// eDataMappingVarNames.powermonitor_InputField_r_EnergySupplied: 				st_Variable:= IotExtractType(monitor.powermonitor.InputField.r_EnergySupplied, 0, 0); 
// eDataMappingVarNames.powermonitor_InputField_ar_THD_AVG: 				st_Variable:= IotExtractType(monitor.powermonitor.InputField.ar_THD[0], 1, 0); 
// eDataMappingVarNames.powermonitor_InputField_ar_THD_L1: 				st_Variable:= IotExtractType(monitor.powermonitor.InputField.ar_THD[1], 1, 0); 
// eDataMappingVarNames.powermonitor_InputField_ar_THD_L2: 				st_Variable:= IotExtractType(monitor.powermonitor.InputField.ar_THD[2], 1, 0); 
// eDataMappingVarNames.powermonitor_InputField_ar_THD_L3: 				st_Variable:= IotExtractType(monitor.powermonitor.InputField.ar_THD[3], 1, 0); 
// eDataMappingVarNames.powermonitor_InputField_ar_PowerFactor_AVG: 				st_Variable:= IotExtractType(monitor.powermonitor.InputField.ar_PowerFactor[0], 2, 0); 
// eDataMappingVarNames.powermonitor_InputField_ar_PowerFactor_L1: 				st_Variable:= IotExtractType(monitor.powermonitor.InputField.ar_PowerFactor[1], 2, 0); 
// eDataMappingVarNames.powermonitor_InputField_ar_PowerFactor_L2: 				st_Variable:= IotExtractType(monitor.powermonitor.InputField.ar_PowerFactor[2], 2, 0); 
// eDataMappingVarNames.powermonitor_InputField_ar_PowerFactor_L3: 				st_Variable:= IotExtractType(monitor.powermonitor.InputField.ar_PowerFactor[3], 2, 0); 
// eDataMappingVarNames.powermonitor_InputField_ar_Current_AVG: 				st_Variable:= IotExtractType(monitor.powermonitor.InputField.ar_Current[0], 0, 1); 
// eDataMappingVarNames.powermonitor_InputField_ar_Current_L1: 				st_Variable:= IotExtractType(monitor.powermonitor.InputField.ar_Current[1], 0, 1); 
// eDataMappingVarNames.powermonitor_InputField_ar_Current_L2: 				st_Variable:= IotExtractType(monitor.powermonitor.InputField.ar_Current[2], 0, 1); 
// eDataMappingVarNames.powermonitor_InputField_ar_Current_L3: 				st_Variable:= IotExtractType(monitor.powermonitor.InputField.ar_Current[3], 0, 1); 
// eDataMappingVarNames.powermonitor_InputField_ar_Current_N: 					st_Variable:= IotExtractType(monitor.powermonitor.InputField.ar_Current[4], 0, 1); 
// eDataMappingVarNames.powermonitor_InputField_r_CurrentUnbalance: 				st_Variable:= IotExtractType(monitor.powermonitor.InputField.r_CurrentUnbalance, 1, 0); 
// eDataMappingVarNames.powermonitor_InputField_e_ACrotationStatus: 				st_Variable:= IotExtractType(monitor.powermonitor.InputField.e_ACrotationStatus, 0, 0); 
// eDataMappingVarNames.powermonitor_InputField_ar_PhaseVoltage_AVG: 				st_Variable:= IotExtractType(monitor.powermonitor.InputField.ar_PhaseVoltage[0], 1, 1); 
// eDataMappingVarNames.powermonitor_InputField_ar_PhaseVoltage_L1: 				st_Variable:= IotExtractType(monitor.powermonitor.InputField.ar_PhaseVoltage[1], 1, 1); 
// eDataMappingVarNames.powermonitor_InputField_ar_PhaseVoltage_L2: 				st_Variable:= IotExtractType(monitor.powermonitor.InputField.ar_PhaseVoltage[2], 1, 1); 
// eDataMappingVarNames.powermonitor_InputField_ar_PhaseVoltage_L3: 				st_Variable:= IotExtractType(monitor.powermonitor.InputField.ar_PhaseVoltage[3], 1, 1); 
// eDataMappingVarNames.powermonitor_InputField_ar_LineVoltage_AVG: 				st_Variable:= IotExtractType(monitor.powermonitor.InputField.ar_LineVoltage[0], 1, 1); 
// eDataMappingVarNames.powermonitor_InputField_ar_LineVoltage_L1: 				st_Variable:= IotExtractType(monitor.powermonitor.InputField.ar_LineVoltage[1], 1, 1); 
// eDataMappingVarNames.powermonitor_InputField_ar_LineVoltage_L2: 				st_Variable:= IotExtractType(monitor.powermonitor.InputField.ar_LineVoltage[2], 1, 1); 
// eDataMappingVarNames.powermonitor_InputField_ar_LineVoltage_L3: 				st_Variable:= IotExtractType(monitor.powermonitor.InputField.ar_LineVoltage[3], 1, 1); 
// eDataMappingVarNames.powermonitor_InputField_li_TimeVoltZeroCrossup: 				st_Variable:= IotExtractType(monitor.powermonitor.InputField.li_TimeVoltZeroCrossup, 0, 0); 
// eDataMappingVarNames.powermonitor_InputField_ar_Frequency_AVG: 				st_Variable:= IotExtractType(monitor.powermonitor.InputField.ar_Frequency[0], 2, 1); 
// eDataMappingVarNames.powermonitor_InputField_ar_Frequency_L1: 				st_Variable:= IotExtractType(monitor.powermonitor.InputField.ar_Frequency[1], 2, 1); 
// eDataMappingVarNames.powermonitor_InputField_ar_Frequency_L2: 				st_Variable:= IotExtractType(monitor.powermonitor.InputField.ar_Frequency[2], 2, 1); 
// eDataMappingVarNames.powermonitor_InputField_ar_Frequency_L3: 				st_Variable:= IotExtractType(monitor.powermonitor.InputField.ar_Frequency[3], 2, 1); 
// eDataMappingVarNames.powermonitor_InputField_r_VoltageUnbalance: 				st_Variable:= IotExtractType(monitor.powermonitor.InputField.r_VoltageUnbalance, 1, 0); 
// eDataMappingVarNames.powermonitor_InputField_r_loadshare: 				st_Variable:= IotExtractType(monitor.powermonitor.InputField.r_loadshare, 1, 0); 
// eDataMappingVarNames.powermonitor_InputField_Powerlock_1_ar_ApparentPower_AVG: 				st_Variable:= IotExtractType(monitor.powermonitor.InputField.Powerlock[1].ar_ApparentPower[0], 0, 0); 
// eDataMappingVarNames.powermonitor_InputField_Powerlock_2_ar_ApparentPower_AVG: 				st_Variable:= IotExtractType(monitor.powermonitor.InputField.Powerlock[2].ar_ApparentPower[0], 0, 0); 
// eDataMappingVarNames.powermonitor_InputField_Powerlock_1_ar_ApparentPower_L1: 				st_Variable:= IotExtractType(monitor.powermonitor.InputField.Powerlock[1].ar_ApparentPower[1], 0, 0); 
// eDataMappingVarNames.powermonitor_InputField_Powerlock_2_ar_ApparentPower_L1: 				st_Variable:= IotExtractType(monitor.powermonitor.InputField.Powerlock[2].ar_ApparentPower[1], 0, 0); 
// eDataMappingVarNames.powermonitor_InputField_Powerlock_1_ar_ApparentPower_L2: 				st_Variable:= IotExtractType(monitor.powermonitor.InputField.Powerlock[1].ar_ApparentPower[2], 0, 0); 
// eDataMappingVarNames.powermonitor_InputField_Powerlock_2_ar_ApparentPower_L2: 				st_Variable:= IotExtractType(monitor.powermonitor.InputField.Powerlock[2].ar_ApparentPower[2], 0, 0); 
// eDataMappingVarNames.powermonitor_InputField_Powerlock_1_ar_ApparentPower_L3: 				st_Variable:= IotExtractType(monitor.powermonitor.InputField.Powerlock[1].ar_ApparentPower[3], 0, 0); 
// eDataMappingVarNames.powermonitor_InputField_Powerlock_2_ar_ApparentPower_L3: 				st_Variable:= IotExtractType(monitor.powermonitor.InputField.Powerlock[2].ar_ApparentPower[3], 0, 0); 
// eDataMappingVarNames.powermonitor_InputField_Powerlock_1_ar_ReactivePower_AVG: 				st_Variable:= IotExtractType(monitor.powermonitor.InputField.Powerlock[1].ar_ReactivePower[0], 0, 0); 
// eDataMappingVarNames.powermonitor_InputField_Powerlock_2_ar_ReactivePower_AVG: 				st_Variable:= IotExtractType(monitor.powermonitor.InputField.Powerlock[2].ar_ReactivePower[0], 0, 0); 
// eDataMappingVarNames.powermonitor_InputField_Powerlock_1_ar_ReactivePower_L1: 				st_Variable:= IotExtractType(monitor.powermonitor.InputField.Powerlock[1].ar_ReactivePower[1], 0, 0); 
// eDataMappingVarNames.powermonitor_InputField_Powerlock_2_ar_ReactivePower_L1: 				st_Variable:= IotExtractType(monitor.powermonitor.InputField.Powerlock[2].ar_ReactivePower[1], 0, 0); 
// eDataMappingVarNames.powermonitor_InputField_Powerlock_1_ar_ReactivePower_L2: 				st_Variable:= IotExtractType(monitor.powermonitor.InputField.Powerlock[1].ar_ReactivePower[2], 0, 0); 
// eDataMappingVarNames.powermonitor_InputField_Powerlock_2_ar_ReactivePower_L2: 				st_Variable:= IotExtractType(monitor.powermonitor.InputField.Powerlock[2].ar_ReactivePower[2], 0, 0); 
// eDataMappingVarNames.powermonitor_InputField_Powerlock_1_ar_ReactivePower_L3: 				st_Variable:= IotExtractType(monitor.powermonitor.InputField.Powerlock[1].ar_ReactivePower[3], 0, 0); 
// eDataMappingVarNames.powermonitor_InputField_Powerlock_2_ar_ReactivePower_L3: 				st_Variable:= IotExtractType(monitor.powermonitor.InputField.Powerlock[2].ar_ReactivePower[3], 0, 0); 
// eDataMappingVarNames.powermonitor_InputField_Powerlock_1_ar_ActivePower_AVG: 				st_Variable:= IotExtractType(monitor.powermonitor.InputField.Powerlock[1].ar_ActivePower[0]	, 0, 0); 
// eDataMappingVarNames.powermonitor_InputField_Powerlock_2_ar_ActivePower_AVG: 				st_Variable:= IotExtractType(monitor.powermonitor.InputField.Powerlock[2].ar_ActivePower[0]	, 0, 0); 
// eDataMappingVarNames.powermonitor_InputField_Powerlock_1_ar_ActivePower_L1: 				st_Variable:= IotExtractType(monitor.powermonitor.InputField.Powerlock[1].ar_ActivePower[1]	, 0, 0); 
// eDataMappingVarNames.powermonitor_InputField_Powerlock_2_ar_ActivePower_L1: 				st_Variable:= IotExtractType(monitor.powermonitor.InputField.Powerlock[2].ar_ActivePower[1]	, 0, 0); 
// eDataMappingVarNames.powermonitor_InputField_Powerlock_1_ar_ActivePower_L2: 				st_Variable:= IotExtractType(monitor.powermonitor.InputField.Powerlock[1].ar_ActivePower[2]	, 0, 0); 
// eDataMappingVarNames.powermonitor_InputField_Powerlock_2_ar_ActivePower_L2: 				st_Variable:= IotExtractType(monitor.powermonitor.InputField.Powerlock[2].ar_ActivePower[2]	, 0, 0); 
// eDataMappingVarNames.powermonitor_InputField_Powerlock_1_ar_ActivePower_L3: 				st_Variable:= IotExtractType(monitor.powermonitor.InputField.Powerlock[1].ar_ActivePower[3]	, 0, 0); 
// eDataMappingVarNames.powermonitor_InputField_Powerlock_2_ar_ActivePower_L3: 				st_Variable:= IotExtractType(monitor.powermonitor.InputField.Powerlock[2].ar_ActivePower[3]	, 0, 0); 
// eDataMappingVarNames.powermonitor_InputField_Powerlock_1_r_EnergyConsumed: 				st_Variable:= IotExtractType(monitor.powermonitor.InputField.Powerlock[1].r_EnergyConsumed, 0, 	0); 
// eDataMappingVarNames.powermonitor_InputField_Powerlock_2_r_EnergyConsumed: 				st_Variable:= IotExtractType(monitor.powermonitor.InputField.Powerlock[2].r_EnergyConsumed, 0, 	0); 
// eDataMappingVarNames.powermonitor_InputField_Powerlock_1_r_EnergySupplied: 				st_Variable:= IotExtractType(monitor.powermonitor.InputField.Powerlock[1].r_EnergySupplied, 0, 	0); 
// eDataMappingVarNames.powermonitor_InputField_Powerlock_2_r_EnergySupplied: 				st_Variable:= IotExtractType(monitor.powermonitor.InputField.Powerlock[2].r_EnergySupplied, 0, 	0); 
// eDataMappingVarNames.powermonitor_InputField_Powerlock_1_ar_THD_AVG: 				st_Variable:= IotExtractType(monitor.powermonitor.InputField.Powerlock[1].ar_THD[0], 0, 0);        	
// eDataMappingVarNames.powermonitor_InputField_Powerlock_2_ar_THD_AVG: 				st_Variable:= IotExtractType(monitor.powermonitor.InputField.Powerlock[2].ar_THD[0], 0, 0);        	
// eDataMappingVarNames.powermonitor_InputField_Powerlock_1_ar_THD_L1: 				st_Variable:= IotExtractType(monitor.powermonitor.InputField.Powerlock[1].ar_THD[1], 0, 0);        	
// eDataMappingVarNames.powermonitor_InputField_Powerlock_2_ar_THD_L1: 				st_Variable:= IotExtractType(monitor.powermonitor.InputField.Powerlock[2].ar_THD[1], 0, 0);        	
// eDataMappingVarNames.powermonitor_InputField_Powerlock_1_ar_THD_L2: 				st_Variable:= IotExtractType(monitor.powermonitor.InputField.Powerlock[1].ar_THD[2], 0, 0);        	
// eDataMappingVarNames.powermonitor_InputField_Powerlock_2_ar_THD_L2: 				st_Variable:= IotExtractType(monitor.powermonitor.InputField.Powerlock[2].ar_THD[2], 0, 0);        	
// eDataMappingVarNames.powermonitor_InputField_Powerlock_1_ar_THD_L3: 				st_Variable:= IotExtractType(monitor.powermonitor.InputField.Powerlock[1].ar_THD[3], 0, 0);        	
// eDataMappingVarNames.powermonitor_InputField_Powerlock_2_ar_THD_L3: 				st_Variable:= IotExtractType(monitor.powermonitor.InputField.Powerlock[2].ar_THD[3], 0, 0);        	
// eDataMappingVarNames.powermonitor_InputField_Powerlock_1_ar_PowerFactor_AVG: 				st_Variable:= IotExtractType(monitor.powermonitor.InputField.Powerlock[1].ar_PowerFactor[0]	, 2, 0); 
// eDataMappingVarNames.powermonitor_InputField_Powerlock_2_ar_PowerFactor_AVG: 				st_Variable:= IotExtractType(monitor.powermonitor.InputField.Powerlock[2].ar_PowerFactor[0]	, 2, 0); 
// eDataMappingVarNames.powermonitor_InputField_Powerlock_1_ar_PowerFactor_L1: 				st_Variable:= IotExtractType(monitor.powermonitor.InputField.Powerlock[1].ar_PowerFactor[1]	, 2, 0); 
// eDataMappingVarNames.powermonitor_InputField_Powerlock_2_ar_PowerFactor_L1: 				st_Variable:= IotExtractType(monitor.powermonitor.InputField.Powerlock[2].ar_PowerFactor[1]	, 2, 0); 
// eDataMappingVarNames.powermonitor_InputField_Powerlock_1_ar_PowerFactor_L2: 				st_Variable:= IotExtractType(monitor.powermonitor.InputField.Powerlock[1].ar_PowerFactor[2]	, 2, 0); 
// eDataMappingVarNames.powermonitor_InputField_Powerlock_2_ar_PowerFactor_L2: 				st_Variable:= IotExtractType(monitor.powermonitor.InputField.Powerlock[2].ar_PowerFactor[2]	, 2, 0); 
// eDataMappingVarNames.powermonitor_InputField_Powerlock_1_ar_PowerFactor_L3: 				st_Variable:= IotExtractType(monitor.powermonitor.InputField.Powerlock[1].ar_PowerFactor[3]	, 2, 0); 
// eDataMappingVarNames.powermonitor_InputField_Powerlock_2_ar_PowerFactor_L3: 				st_Variable:= IotExtractType(monitor.powermonitor.InputField.Powerlock[2].ar_PowerFactor[3]	, 2, 0); 
// eDataMappingVarNames.powermonitor_InputField_Powerlock_1_ar_Current_AVG: 				st_Variable:= IotExtractType(monitor.powermonitor.InputField.Powerlock[1].ar_Current[0]			, 1, 1); 
// eDataMappingVarNames.powermonitor_InputField_Powerlock_2_ar_Current_AVG: 				st_Variable:= IotExtractType(monitor.powermonitor.InputField.Powerlock[2].ar_Current[0]			, 1, 1); 
// eDataMappingVarNames.powermonitor_InputField_Powerlock_1_ar_Current_L1: 				st_Variable:= IotExtractType(monitor.powermonitor.InputField.Powerlock[1].ar_Current[1]			, 1, 1); 
// eDataMappingVarNames.powermonitor_InputField_Powerlock_2_ar_Current_L1: 				st_Variable:= IotExtractType(monitor.powermonitor.InputField.Powerlock[2].ar_Current[1]			, 1, 1); 
// eDataMappingVarNames.powermonitor_InputField_Powerlock_1_ar_Current_L2: 				st_Variable:= IotExtractType(monitor.powermonitor.InputField.Powerlock[1].ar_Current[2]			, 1, 1); 
// eDataMappingVarNames.powermonitor_InputField_Powerlock_2_ar_Current_L2: 				st_Variable:= IotExtractType(monitor.powermonitor.InputField.Powerlock[2].ar_Current[2]			, 1, 1); 
// eDataMappingVarNames.powermonitor_InputField_Powerlock_1_ar_Current_L3: 				st_Variable:= IotExtractType(monitor.powermonitor.InputField.Powerlock[1].ar_Current[3]			, 1, 1); 
// eDataMappingVarNames.powermonitor_InputField_Powerlock_2_ar_Current_L3: 				st_Variable:= IotExtractType(monitor.powermonitor.InputField.Powerlock[2].ar_Current[3]			, 1, 1); 
// eDataMappingVarNames.powermonitor_InputField_Powerlock_1_ar_Current_N: 				st_Variable:= IotExtractType(monitor.powermonitor.InputField.Powerlock[1].ar_Current[4], 1, 1); 
// eDataMappingVarNames.powermonitor_InputField_Powerlock_2_ar_Current_N: 				st_Variable:= IotExtractType(monitor.powermonitor.InputField.Powerlock[2].ar_Current[4], 1, 1); 
// eDataMappingVarNames.powermonitor_InputField_Powerlock_1_r_CurrentUnbalance: 				st_Variable:= IotExtractType(monitor.powermonitor.InputField.Powerlock[1].r_CurrentUnbalance, 0, 0); 
// eDataMappingVarNames.powermonitor_InputField_Powerlock_2_r_CurrentUnbalance: 				st_Variable:= IotExtractType(monitor.powermonitor.InputField.Powerlock[2].r_CurrentUnbalance, 0, 0); 
// eDataMappingVarNames.powermonitor_OutputField_ar_ApparentPower_AVG: 				st_Variable:= IotExtractType(monitor.powermonitor.OutputField.ar_ApparentPower[0]	, 1, 1); 
// eDataMappingVarNames.powermonitor_OutputField_ar_ApparentPower_L1: 				st_Variable:= IotExtractType(monitor.powermonitor.OutputField.ar_ApparentPower[1]		, 1, 1); 
// eDataMappingVarNames.powermonitor_OutputField_ar_ApparentPower_L2: 				st_Variable:= IotExtractType(monitor.powermonitor.OutputField.ar_ApparentPower[2]		, 1, 1); 
// eDataMappingVarNames.powermonitor_OutputField_ar_ApparentPower_L3: 				st_Variable:= IotExtractType(monitor.powermonitor.OutputField.ar_ApparentPower[3]		, 1, 1); 
// eDataMappingVarNames.powermonitor_OutputField_ar_ReactivePower_AVG: 				st_Variable:= IotExtractType(monitor.powermonitor.OutputField.ar_ReactivePower[0]	, 1, 1); 
// eDataMappingVarNames.powermonitor_OutputField_ar_ReactivePower_L1: 				st_Variable:= IotExtractType(monitor.powermonitor.OutputField.ar_ReactivePower[1]		, 1, 1); 
// eDataMappingVarNames.powermonitor_OutputField_ar_ReactivePower_L2: 				st_Variable:= IotExtractType(monitor.powermonitor.OutputField.ar_ReactivePower[2]		, 1, 1); 
// eDataMappingVarNames.powermonitor_OutputField_ar_ReactivePower_L3: 				st_Variable:= IotExtractType(monitor.powermonitor.OutputField.ar_ReactivePower[3]		, 1, 1); 
// eDataMappingVarNames.powermonitor_OutputField_ar_ActivePower_AVG: 				st_Variable:= IotExtractType(monitor.powermonitor.OutputField.ar_ActivePower[0]			, 1, 1); 
// eDataMappingVarNames.powermonitor_OutputField_ar_ActivePower_L1: 				st_Variable:= IotExtractType(monitor.powermonitor.OutputField.ar_ActivePower[1]			, 1, 1); 
// eDataMappingVarNames.powermonitor_OutputField_ar_ActivePower_L2: 				st_Variable:= IotExtractType(monitor.powermonitor.OutputField.ar_ActivePower[2]			, 1, 1); 
// eDataMappingVarNames.powermonitor_OutputField_ar_ActivePower_L3: 				st_Variable:= IotExtractType(monitor.powermonitor.OutputField.ar_ActivePower[3]			, 1, 1); 
// eDataMappingVarNames.powermonitor_OutputField_r_EnergyConsumed: 				st_Variable:= IotExtractType(monitor.powermonitor.OutputField.r_EnergyConsumed, 0, 0); 
// eDataMappingVarNames.powermonitor_OutputField_r_EnergySupplied: 				st_Variable:= IotExtractType(monitor.powermonitor.OutputField.r_EnergySupplied, 0, 0); 
// eDataMappingVarNames.powermonitor_OutputField_ar_THD_AVG: 				st_Variable:= IotExtractType(monitor.powermonitor.OutputField.ar_THD[0], 1, 0); 
// eDataMappingVarNames.powermonitor_OutputField_ar_THD_L1: 				st_Variable:= IotExtractType(monitor.powermonitor.OutputField.ar_THD[1], 1, 0); 
// eDataMappingVarNames.powermonitor_OutputField_ar_THD_L2: 				st_Variable:= IotExtractType(monitor.powermonitor.OutputField.ar_THD[2], 1, 0); 
// eDataMappingVarNames.powermonitor_OutputField_ar_THD_L3: 				st_Variable:= IotExtractType(monitor.powermonitor.OutputField.ar_THD[3], 1, 0); 
// eDataMappingVarNames.powermonitor_OutputField_ar_PowerFactor_AVG: 				st_Variable:= IotExtractType(monitor.powermonitor.OutputField.ar_PowerFactor[0], 2, 0); 
// eDataMappingVarNames.powermonitor_OutputField_ar_PowerFactor_L1: 				st_Variable:= IotExtractType(monitor.powermonitor.OutputField.ar_PowerFactor[1], 2, 0); 
// eDataMappingVarNames.powermonitor_OutputField_ar_PowerFactor_L2: 				st_Variable:= IotExtractType(monitor.powermonitor.OutputField.ar_PowerFactor[2], 2, 0); 
// eDataMappingVarNames.powermonitor_OutputField_ar_PowerFactor_L3: 				st_Variable:= IotExtractType(monitor.powermonitor.OutputField.ar_PowerFactor[3], 2, 0); 
// eDataMappingVarNames.powermonitor_OutputField_ar_Current_AVG: 				st_Variable:= IotExtractType(monitor.powermonitor.OutputField.ar_Current[0], 1, 1); 
// eDataMappingVarNames.powermonitor_OutputField_ar_Current_L1: 				st_Variable:= IotExtractType(monitor.powermonitor.OutputField.ar_Current[1], 1, 1); 
// eDataMappingVarNames.powermonitor_OutputField_ar_Current_L2: 				st_Variable:= IotExtractType(monitor.powermonitor.OutputField.ar_Current[2], 1, 1); 
// eDataMappingVarNames.powermonitor_OutputField_ar_Current_L3: 				st_Variable:= IotExtractType(monitor.powermonitor.OutputField.ar_Current[3], 1, 1); 
// eDataMappingVarNames.powermonitor_OutputField_ar_Current_N: 				st_Variable:= IotExtractType(monitor.powermonitor.OutputField.ar_Current[4], 1, 1); 
// eDataMappingVarNames.powermonitor_OutputField_r_CurrentUnbalance: 				st_Variable:= IotExtractType(monitor.powermonitor.OutputField.r_CurrentUnbalance, 1, 0); 
// eDataMappingVarNames.powermonitor_OutputField_e_ACrotationStatus: 				st_Variable:= IotExtractType(monitor.powermonitor.OutputField.e_ACrotationStatus, 0, 0); 
// eDataMappingVarNames.powermonitor_OutputField_ar_PhaseVoltage_AVG: 				st_Variable:= IotExtractType(monitor.powermonitor.OutputField.ar_PhaseVoltage[0], 1, 1); 
// eDataMappingVarNames.powermonitor_OutputField_ar_PhaseVoltage_L1: 				st_Variable:= IotExtractType(monitor.powermonitor.OutputField.ar_PhaseVoltage[1], 1, 1); 
// eDataMappingVarNames.powermonitor_OutputField_ar_PhaseVoltage_L2: 				st_Variable:= IotExtractType(monitor.powermonitor.OutputField.ar_PhaseVoltage[2], 1, 1); 
// eDataMappingVarNames.powermonitor_OutputField_ar_PhaseVoltage_L3: 				st_Variable:= IotExtractType(monitor.powermonitor.OutputField.ar_PhaseVoltage[3], 1, 1); 
// eDataMappingVarNames.powermonitor_OutputField_ar_LineVoltage_AVG: 				st_Variable:= IotExtractType(monitor.powermonitor.OutputField.ar_LineVoltage[0]	, 1, 1); 
// eDataMappingVarNames.powermonitor_OutputField_ar_LineVoltage_L1: 				st_Variable:= IotExtractType(monitor.powermonitor.OutputField.ar_LineVoltage[1]	, 1, 1); 
// eDataMappingVarNames.powermonitor_OutputField_ar_LineVoltage_L2: 				st_Variable:= IotExtractType(monitor.powermonitor.OutputField.ar_LineVoltage[2]	, 1, 1); 
// eDataMappingVarNames.powermonitor_OutputField_ar_LineVoltage_L3: 				st_Variable:= IotExtractType(monitor.powermonitor.OutputField.ar_LineVoltage[3]	, 1, 1); 
// eDataMappingVarNames.powermonitor_OutputField_li_TimeVoltZeroCrossup: 				st_Variable:= IotExtractType(monitor.powermonitor.OutputField.li_TimeVoltZeroCrossup, 0, 0); 
// eDataMappingVarNames.powermonitor_OutputField_ar_Frequency_AVG: 				st_Variable:= IotExtractType(monitor.powermonitor.OutputField.ar_Frequency[0], 2, 1); 
// eDataMappingVarNames.powermonitor_OutputField_ar_Frequency_L1: 				st_Variable:= IotExtractType(monitor.powermonitor.OutputField.ar_Frequency[1], 2, 1); 
// eDataMappingVarNames.powermonitor_OutputField_ar_Frequency_L2: 				st_Variable:= IotExtractType(monitor.powermonitor.OutputField.ar_Frequency[2], 2, 1); 
// eDataMappingVarNames.powermonitor_OutputField_ar_Frequency_L3: 				st_Variable:= IotExtractType(monitor.powermonitor.OutputField.ar_Frequency[3], 2, 1); 
// eDataMappingVarNames.powermonitor_OutputField_r_VoltageUnbalance: 				st_Variable:= IotExtractType(monitor.powermonitor.OutputField.r_VoltageUnbalance, 1, 0); 
// eDataMappingVarNames.powermonitor_OutputField_r_loadshare: 				st_Variable:= IotExtractType(monitor.powermonitor.OutputField.r_loadshare, 1, 0); 
// eDataMappingVarNames.powermonitor_OutputField_Powerlock_1_ar_ApparentPower_AVG: 				st_Variable:= IotExtractType(monitor.powermonitor.OutputField.Powerlock[1].ar_ApparentPower[0]	, 1, 1); 
// eDataMappingVarNames.powermonitor_OutputField_Powerlock_2_ar_ApparentPower_AVG: 				st_Variable:= IotExtractType(monitor.powermonitor.OutputField.Powerlock[2].ar_ApparentPower[0]	, 1, 1); 
// eDataMappingVarNames.powermonitor_OutputField_Powerlock_3_ar_ApparentPower_AVG: 				st_Variable:= IotExtractType(monitor.powermonitor.OutputField.Powerlock[3].ar_ApparentPower[0]	, 1, 1); 
// eDataMappingVarNames.powermonitor_OutputField_Powerlock_1_ar_ApparentPower_L1: 				st_Variable:= IotExtractType(monitor.powermonitor.OutputField.Powerlock[1].ar_ApparentPower[1]		, 1, 1); 
// eDataMappingVarNames.powermonitor_OutputField_Powerlock_2_ar_ApparentPower_L1: 				st_Variable:= IotExtractType(monitor.powermonitor.OutputField.Powerlock[2].ar_ApparentPower[1]		, 1, 1); 
// eDataMappingVarNames.powermonitor_OutputField_Powerlock_3_ar_ApparentPower_L1: 				st_Variable:= IotExtractType(monitor.powermonitor.OutputField.Powerlock[3].ar_ApparentPower[1]		, 1, 1); 
// eDataMappingVarNames.powermonitor_OutputField_Powerlock_1_ar_ApparentPower_L2: 				st_Variable:= IotExtractType(monitor.powermonitor.OutputField.Powerlock[1].ar_ApparentPower[2]		, 1, 1); 
// eDataMappingVarNames.powermonitor_OutputField_Powerlock_2_ar_ApparentPower_L2: 				st_Variable:= IotExtractType(monitor.powermonitor.OutputField.Powerlock[2].ar_ApparentPower[2]		, 1, 1); 
// eDataMappingVarNames.powermonitor_OutputField_Powerlock_3_ar_ApparentPower_L2: 				st_Variable:= IotExtractType(monitor.powermonitor.OutputField.Powerlock[3].ar_ApparentPower[2]		, 1, 1); 
// eDataMappingVarNames.powermonitor_OutputField_Powerlock_1_ar_ApparentPower_L3: 				st_Variable:= IotExtractType(monitor.powermonitor.OutputField.Powerlock[1].ar_ApparentPower[3]		, 1, 1); 
// eDataMappingVarNames.powermonitor_OutputField_Powerlock_2_ar_ApparentPower_L3: 				st_Variable:= IotExtractType(monitor.powermonitor.OutputField.Powerlock[2].ar_ApparentPower[3]		, 1, 1); 
// eDataMappingVarNames.powermonitor_OutputField_Powerlock_3_ar_ApparentPower_L3: 				st_Variable:= IotExtractType(monitor.powermonitor.OutputField.Powerlock[3].ar_ApparentPower[3]		, 1, 1); 
// eDataMappingVarNames.powermonitor_OutputField_Powerlock_1_ar_ReactivePower_AVG: 				st_Variable:= IotExtractType(monitor.powermonitor.OutputField.Powerlock[1].ar_ReactivePower[0]	, 1, 1); 
// eDataMappingVarNames.powermonitor_OutputField_Powerlock_2_ar_ReactivePower_AVG: 				st_Variable:= IotExtractType(monitor.powermonitor.OutputField.Powerlock[2].ar_ReactivePower[0]	, 1, 1); 
// eDataMappingVarNames.powermonitor_OutputField_Powerlock_3_ar_ReactivePower_AVG: 				st_Variable:= IotExtractType(monitor.powermonitor.OutputField.Powerlock[3].ar_ReactivePower[0]	, 1, 1); 
// eDataMappingVarNames.powermonitor_OutputField_Powerlock_1_ar_ReactivePower_L1: 				st_Variable:= IotExtractType(monitor.powermonitor.OutputField.Powerlock[1].ar_ReactivePower[1]		, 1, 1); 
// eDataMappingVarNames.powermonitor_OutputField_Powerlock_2_ar_ReactivePower_L1: 				st_Variable:= IotExtractType(monitor.powermonitor.OutputField.Powerlock[2].ar_ReactivePower[1]		, 1, 1); 
// eDataMappingVarNames.powermonitor_OutputField_Powerlock_3_ar_ReactivePower_L1: 				st_Variable:= IotExtractType(monitor.powermonitor.OutputField.Powerlock[3].ar_ReactivePower[1]		, 1, 1); 
// eDataMappingVarNames.powermonitor_OutputField_Powerlock_1_ar_ReactivePower_L2: 				st_Variable:= IotExtractType(monitor.powermonitor.OutputField.Powerlock[1].ar_ReactivePower[2]		, 1, 1); 
// eDataMappingVarNames.powermonitor_OutputField_Powerlock_2_ar_ReactivePower_L2: 				st_Variable:= IotExtractType(monitor.powermonitor.OutputField.Powerlock[2].ar_ReactivePower[2]		, 1, 1); 
// eDataMappingVarNames.powermonitor_OutputField_Powerlock_3_ar_ReactivePower_L2: 				st_Variable:= IotExtractType(monitor.powermonitor.OutputField.Powerlock[3].ar_ReactivePower[2]		, 1, 1); 
// eDataMappingVarNames.powermonitor_OutputField_Powerlock_1_ar_ReactivePower_L3: 				st_Variable:= IotExtractType(monitor.powermonitor.OutputField.Powerlock[1].ar_ReactivePower[3]		, 1, 1); 
// eDataMappingVarNames.powermonitor_OutputField_Powerlock_2_ar_ReactivePower_L3: 				st_Variable:= IotExtractType(monitor.powermonitor.OutputField.Powerlock[2].ar_ReactivePower[3]		, 1, 1); 
// eDataMappingVarNames.powermonitor_OutputField_Powerlock_3_ar_ReactivePower_L3: 				st_Variable:= IotExtractType(monitor.powermonitor.OutputField.Powerlock[3].ar_ReactivePower[3]		, 1, 1); 
// eDataMappingVarNames.powermonitor_OutputField_Powerlock_1_ar_ActivePower_AVG: 				st_Variable:= IotExtractType(monitor.powermonitor.OutputField.Powerlock[1].ar_ActivePower[0]		, 1, 1); 
// eDataMappingVarNames.powermonitor_OutputField_Powerlock_2_ar_ActivePower_AVG: 				st_Variable:= IotExtractType(monitor.powermonitor.OutputField.Powerlock[2].ar_ActivePower[0]		, 1, 1); 
// eDataMappingVarNames.powermonitor_OutputField_Powerlock_3_ar_ActivePower_AVG: 				st_Variable:= IotExtractType(monitor.powermonitor.OutputField.Powerlock[3].ar_ActivePower[0]		, 1, 1); 
// eDataMappingVarNames.powermonitor_OutputField_Powerlock_1_ar_ActivePower_L1: 				st_Variable:= IotExtractType(monitor.powermonitor.OutputField.Powerlock[1].ar_ActivePower[1]		, 1, 1); 
// eDataMappingVarNames.powermonitor_OutputField_Powerlock_2_ar_ActivePower_L1: 				st_Variable:= IotExtractType(monitor.powermonitor.OutputField.Powerlock[2].ar_ActivePower[1]		, 1, 1); 
// eDataMappingVarNames.powermonitor_OutputField_Powerlock_3_ar_ActivePower_L1: 				st_Variable:= IotExtractType(monitor.powermonitor.OutputField.Powerlock[3].ar_ActivePower[1]		, 1, 1); 
// eDataMappingVarNames.powermonitor_OutputField_Powerlock_1_ar_ActivePower_L2: 				st_Variable:= IotExtractType(monitor.powermonitor.OutputField.Powerlock[1].ar_ActivePower[2]		, 1, 1); 
// eDataMappingVarNames.powermonitor_OutputField_Powerlock_2_ar_ActivePower_L2: 				st_Variable:= IotExtractType(monitor.powermonitor.OutputField.Powerlock[2].ar_ActivePower[2]		, 1, 1); 
// eDataMappingVarNames.powermonitor_OutputField_Powerlock_3_ar_ActivePower_L2: 				st_Variable:= IotExtractType(monitor.powermonitor.OutputField.Powerlock[3].ar_ActivePower[2]		, 1, 1); 
// eDataMappingVarNames.powermonitor_OutputField_Powerlock_1_ar_ActivePower_L3: 				st_Variable:= IotExtractType(monitor.powermonitor.OutputField.Powerlock[1].ar_ActivePower[3]		, 1, 1); 
// eDataMappingVarNames.powermonitor_OutputField_Powerlock_2_ar_ActivePower_L3: 				st_Variable:= IotExtractType(monitor.powermonitor.OutputField.Powerlock[2].ar_ActivePower[3]		, 1, 1); 
// eDataMappingVarNames.powermonitor_OutputField_Powerlock_3_ar_ActivePower_L3: 				st_Variable:= IotExtractType(monitor.powermonitor.OutputField.Powerlock[3].ar_ActivePower[3]		, 1, 1); 
// eDataMappingVarNames.powermonitor_OutputField_Powerlock_1_r_EnergyConsumed: 				st_Variable:= IotExtractType(monitor.powermonitor.OutputField.Powerlock[1].r_EnergyConsumed, 0, 0); 
// eDataMappingVarNames.powermonitor_OutputField_Powerlock_2_r_EnergyConsumed: 				st_Variable:= IotExtractType(monitor.powermonitor.OutputField.Powerlock[2].r_EnergyConsumed, 0, 0); 
// eDataMappingVarNames.powermonitor_OutputField_Powerlock_3_r_EnergyConsumed: 				st_Variable:= IotExtractType(monitor.powermonitor.OutputField.Powerlock[3].r_EnergyConsumed, 0, 0); 
// eDataMappingVarNames.powermonitor_OutputField_Powerlock_1_r_EnergySupplied: 				st_Variable:= IotExtractType(monitor.powermonitor.OutputField.Powerlock[1].r_EnergySupplied, 0, 0); 
// eDataMappingVarNames.powermonitor_OutputField_Powerlock_2_r_EnergySupplied: 				st_Variable:= IotExtractType(monitor.powermonitor.OutputField.Powerlock[2].r_EnergySupplied, 0, 0); 
// eDataMappingVarNames.powermonitor_OutputField_Powerlock_3_r_EnergySupplied: 				st_Variable:= IotExtractType(monitor.powermonitor.OutputField.Powerlock[3].r_EnergySupplied, 0, 0); 
// eDataMappingVarNames.powermonitor_OutputField_Powerlock_1_ar_THD_AVG: 				st_Variable:= IotExtractType(monitor.powermonitor.OutputField.Powerlock[1].ar_THD[0]						, 1, 0); 
// eDataMappingVarNames.powermonitor_OutputField_Powerlock_2_ar_THD_AVG: 				st_Variable:= IotExtractType(monitor.powermonitor.OutputField.Powerlock[2].ar_THD[0]						, 1, 0); 
// eDataMappingVarNames.powermonitor_OutputField_Powerlock_3_ar_THD_AVG: 				st_Variable:= IotExtractType(monitor.powermonitor.OutputField.Powerlock[3].ar_THD[0]						, 1, 0); 
// eDataMappingVarNames.powermonitor_OutputField_Powerlock_1_ar_THD_L1: 				st_Variable:= IotExtractType(monitor.powermonitor.OutputField.Powerlock[1].ar_THD[1]						, 1, 0); 
// eDataMappingVarNames.powermonitor_OutputField_Powerlock_2_ar_THD_L1: 				st_Variable:= IotExtractType(monitor.powermonitor.OutputField.Powerlock[2].ar_THD[1]						, 1, 0); 
// eDataMappingVarNames.powermonitor_OutputField_Powerlock_3_ar_THD_L1: 				st_Variable:= IotExtractType(monitor.powermonitor.OutputField.Powerlock[3].ar_THD[1]						, 1, 0); 
// eDataMappingVarNames.powermonitor_OutputField_Powerlock_1_ar_THD_L2: 				st_Variable:= IotExtractType(monitor.powermonitor.OutputField.Powerlock[1].ar_THD[2]						, 1, 0); 
// eDataMappingVarNames.powermonitor_OutputField_Powerlock_2_ar_THD_L2: 				st_Variable:= IotExtractType(monitor.powermonitor.OutputField.Powerlock[2].ar_THD[2]						, 1, 0); 
// eDataMappingVarNames.powermonitor_OutputField_Powerlock_3_ar_THD_L2: 				st_Variable:= IotExtractType(monitor.powermonitor.OutputField.Powerlock[3].ar_THD[2]						, 1, 0); 
// eDataMappingVarNames.powermonitor_OutputField_Powerlock_1_ar_THD_L3: 				st_Variable:= IotExtractType(monitor.powermonitor.OutputField.Powerlock[1].ar_THD[3]						, 1, 0); 
// eDataMappingVarNames.powermonitor_OutputField_Powerlock_2_ar_THD_L3: 				st_Variable:= IotExtractType(monitor.powermonitor.OutputField.Powerlock[2].ar_THD[3]						, 1, 0); 
// eDataMappingVarNames.powermonitor_OutputField_Powerlock_3_ar_THD_L3: 				st_Variable:= IotExtractType(monitor.powermonitor.OutputField.Powerlock[3].ar_THD[3]						, 1, 0); 
// eDataMappingVarNames.powermonitor_OutputField_Powerlock_1_ar_PowerFactor_AVG: 				st_Variable:= IotExtractType(monitor.powermonitor.OutputField.Powerlock[1].ar_PowerFactor[0]		, 2, 0); 
// eDataMappingVarNames.powermonitor_OutputField_Powerlock_2_ar_PowerFactor_AVG: 				st_Variable:= IotExtractType(monitor.powermonitor.OutputField.Powerlock[2].ar_PowerFactor[0]		, 2, 0); 
// eDataMappingVarNames.powermonitor_OutputField_Powerlock_3_ar_PowerFactor_AVG: 				st_Variable:= IotExtractType(monitor.powermonitor.OutputField.Powerlock[3].ar_PowerFactor[0]		, 2, 0); 
// eDataMappingVarNames.powermonitor_OutputField_Powerlock_1_ar_PowerFactor_L1: 				st_Variable:= IotExtractType(monitor.powermonitor.OutputField.Powerlock[1].ar_PowerFactor[1]		, 2, 0); 
// eDataMappingVarNames.powermonitor_OutputField_Powerlock_2_ar_PowerFactor_L1: 				st_Variable:= IotExtractType(monitor.powermonitor.OutputField.Powerlock[2].ar_PowerFactor[1]		, 2, 0); 
// eDataMappingVarNames.powermonitor_OutputField_Powerlock_3_ar_PowerFactor_L1: 				st_Variable:= IotExtractType(monitor.powermonitor.OutputField.Powerlock[3].ar_PowerFactor[1]		, 2, 0); 
// eDataMappingVarNames.powermonitor_OutputField_Powerlock_1_ar_PowerFactor_L2: 				st_Variable:= IotExtractType(monitor.powermonitor.OutputField.Powerlock[1].ar_PowerFactor[2]		, 2, 0); 
// eDataMappingVarNames.powermonitor_OutputField_Powerlock_2_ar_PowerFactor_L2: 				st_Variable:= IotExtractType(monitor.powermonitor.OutputField.Powerlock[2].ar_PowerFactor[2]		, 2, 0); 
// eDataMappingVarNames.powermonitor_OutputField_Powerlock_3_ar_PowerFactor_L2: 				st_Variable:= IotExtractType(monitor.powermonitor.OutputField.Powerlock[3].ar_PowerFactor[2]		, 2, 0); 
// eDataMappingVarNames.powermonitor_OutputField_Powerlock_1_ar_PowerFactor_L3: 				st_Variable:= IotExtractType(monitor.powermonitor.OutputField.Powerlock[1].ar_PowerFactor[3]		, 2, 0); 
// eDataMappingVarNames.powermonitor_OutputField_Powerlock_2_ar_PowerFactor_L3: 				st_Variable:= IotExtractType(monitor.powermonitor.OutputField.Powerlock[2].ar_PowerFactor[3]		, 2, 0); 
// eDataMappingVarNames.powermonitor_OutputField_Powerlock_3_ar_PowerFactor_L3: 				st_Variable:= IotExtractType(monitor.powermonitor.OutputField.Powerlock[3].ar_PowerFactor[3]		, 2, 0); 
// eDataMappingVarNames.powermonitor_OutputField_Powerlock_1_ar_Current_AVG: 				st_Variable:= IotExtractType(monitor.powermonitor.OutputField.Powerlock[1].ar_Current[0]				, 1, 1); 
// eDataMappingVarNames.powermonitor_OutputField_Powerlock_2_ar_Current_AVG: 				st_Variable:= IotExtractType(monitor.powermonitor.OutputField.Powerlock[2].ar_Current[0]				, 1, 1); 
// eDataMappingVarNames.powermonitor_OutputField_Powerlock_3_ar_Current_AVG: 				st_Variable:= IotExtractType(monitor.powermonitor.OutputField.Powerlock[3].ar_Current[0]				, 1, 1); 
// eDataMappingVarNames.powermonitor_OutputField_Powerlock_1_ar_Current_L1: 				st_Variable:= IotExtractType(monitor.powermonitor.OutputField.Powerlock[1].ar_Current[1]				, 1, 1); 
// eDataMappingVarNames.powermonitor_OutputField_Powerlock_2_ar_Current_L1: 				st_Variable:= IotExtractType(monitor.powermonitor.OutputField.Powerlock[2].ar_Current[1]				, 1, 1); 
// eDataMappingVarNames.powermonitor_OutputField_Powerlock_3_ar_Current_L1: 				st_Variable:= IotExtractType(monitor.powermonitor.OutputField.Powerlock[3].ar_Current[1]				, 1, 1); 
// eDataMappingVarNames.powermonitor_OutputField_Powerlock_1_ar_Current_L2: 				st_Variable:= IotExtractType(monitor.powermonitor.OutputField.Powerlock[1].ar_Current[2]				, 1, 1); 
// eDataMappingVarNames.powermonitor_OutputField_Powerlock_2_ar_Current_L2: 				st_Variable:= IotExtractType(monitor.powermonitor.OutputField.Powerlock[2].ar_Current[2]				, 1, 1); 
// eDataMappingVarNames.powermonitor_OutputField_Powerlock_3_ar_Current_L2: 				st_Variable:= IotExtractType(monitor.powermonitor.OutputField.Powerlock[3].ar_Current[2]				, 1, 1); 
// eDataMappingVarNames.powermonitor_OutputField_Powerlock_1_ar_Current_L3: 				st_Variable:= IotExtractType(monitor.powermonitor.OutputField.Powerlock[1].ar_Current[3]				, 1, 1); 
// eDataMappingVarNames.powermonitor_OutputField_Powerlock_2_ar_Current_L3: 				st_Variable:= IotExtractType(monitor.powermonitor.OutputField.Powerlock[2].ar_Current[3]				, 1, 1); 
// eDataMappingVarNames.powermonitor_OutputField_Powerlock_3_ar_Current_L3: 				st_Variable:= IotExtractType(monitor.powermonitor.OutputField.Powerlock[3].ar_Current[3]				, 1, 1); 
// eDataMappingVarNames.powermonitor_OutputField_Powerlock_1_ar_Current_N: 				st_Variable:= IotExtractType(monitor.powermonitor.OutputField.Powerlock[1].ar_Current[4]				, 1, 1); 
// eDataMappingVarNames.powermonitor_OutputField_Powerlock_2_ar_Current_N: 				st_Variable:= IotExtractType(monitor.powermonitor.OutputField.Powerlock[2].ar_Current[4]				, 1, 1); 
// eDataMappingVarNames.powermonitor_OutputField_Powerlock_3_ar_Current_N: 				st_Variable:= IotExtractType(monitor.powermonitor.OutputField.Powerlock[3].ar_Current[4]				, 1, 1); 
// eDataMappingVarNames.powermonitor_OutputField_Powerlock_1_r_CurrentUnbalance: 				st_Variable:= IotExtractType(monitor.powermonitor.OutputField.Powerlock[1].r_CurrentUnbalance, 0, 0); 
// eDataMappingVarNames.powermonitor_OutputField_Powerlock_2_r_CurrentUnbalance: 				st_Variable:= IotExtractType(monitor.powermonitor.OutputField.Powerlock[2].r_CurrentUnbalance, 0, 0); 
// eDataMappingVarNames.powermonitor_OutputField_Powerlock_3_r_CurrentUnbalance: 				st_Variable:= IotExtractType(monitor.powermonitor.OutputField.Powerlock[3].r_CurrentUnbalance, 0, 0); 
// eDataMappingVarNames.powermonitor_InternalSupply_ar_ApparentPower_AVG: 				st_Variable:= IotExtractType(monitor.powermonitor.InternalSupply.ar_ApparentPower[0], 2, 0); 
// eDataMappingVarNames.powermonitor_InternalSupply_ar_ApparentPower_L1: 				st_Variable:= IotExtractType(monitor.powermonitor.InternalSupply.ar_ApparentPower[1], 2, 0); 
// eDataMappingVarNames.powermonitor_InternalSupply_ar_ApparentPower_L2: 				st_Variable:= IotExtractType(monitor.powermonitor.InternalSupply.ar_ApparentPower[2], 2, 0); 
// eDataMappingVarNames.powermonitor_InternalSupply_ar_ApparentPower_L3: 				st_Variable:= IotExtractType(monitor.powermonitor.InternalSupply.ar_ApparentPower[3], 2, 0); 
// eDataMappingVarNames.powermonitor_InternalSupply_ar_ReactivePower_AVG: 				st_Variable:= IotExtractType(monitor.powermonitor.InternalSupply.ar_ReactivePower[0], 2, 0); 
// eDataMappingVarNames.powermonitor_InternalSupply_ar_ReactivePower_L1: 				st_Variable:= IotExtractType(monitor.powermonitor.InternalSupply.ar_ReactivePower[1], 2, 0); 
// eDataMappingVarNames.powermonitor_InternalSupply_ar_ReactivePower_L2: 				st_Variable:= IotExtractType(monitor.powermonitor.InternalSupply.ar_ReactivePower[2], 2, 0); 
// eDataMappingVarNames.powermonitor_InternalSupply_ar_ReactivePower_L3: 				st_Variable:= IotExtractType(monitor.powermonitor.InternalSupply.ar_ReactivePower[3], 2, 0); 
// eDataMappingVarNames.powermonitor_InternalSupply_ar_ActivePower_AVG: 				st_Variable:= IotExtractType(monitor.powermonitor.InternalSupply.ar_ActivePower[0], 2, 0); 
// eDataMappingVarNames.powermonitor_InternalSupply_ar_ActivePower_L1: 				st_Variable:= IotExtractType(monitor.powermonitor.InternalSupply.ar_ActivePower[1], 2, 0); 
// eDataMappingVarNames.powermonitor_InternalSupply_ar_ActivePower_L2: 				st_Variable:= IotExtractType(monitor.powermonitor.InternalSupply.ar_ActivePower[2], 2, 0); 
// eDataMappingVarNames.powermonitor_InternalSupply_ar_ActivePower_L3: 				st_Variable:= IotExtractType(monitor.powermonitor.InternalSupply.ar_ActivePower[3], 2, 0); 
// eDataMappingVarNames.powermonitor_InternalSupply_r_EnergyConsumed: 				st_Variable:= IotExtractType(monitor.powermonitor.InternalSupply.r_EnergyConsumed, 0, 0); 
// eDataMappingVarNames.powermonitor_InternalSupply_r_EnergySupplied: 				st_Variable:= IotExtractType(monitor.powermonitor.InternalSupply.r_EnergySupplied, 0, 0); 
// eDataMappingVarNames.powermonitor_InternalSupply_ar_THD_AVG: 				st_Variable:= IotExtractType(monitor.powermonitor.InternalSupply.ar_THD[0], 1, 0); 
// eDataMappingVarNames.powermonitor_InternalSupply_ar_THD_L1: 				st_Variable:= IotExtractType(monitor.powermonitor.InternalSupply.ar_THD[1], 1, 0); 
// eDataMappingVarNames.powermonitor_InternalSupply_ar_THD_L2: 				st_Variable:= IotExtractType(monitor.powermonitor.InternalSupply.ar_THD[2], 1, 0); 
// eDataMappingVarNames.powermonitor_InternalSupply_ar_THD_L3: 				st_Variable:= IotExtractType(monitor.powermonitor.InternalSupply.ar_THD[3], 1, 0); 
// eDataMappingVarNames.powermonitor_InternalSupply_ar_PowerFactor_AVG: 				st_Variable:= IotExtractType(monitor.powermonitor.InternalSupply.ar_PowerFactor[0], 2, 0); 
// eDataMappingVarNames.powermonitor_InternalSupply_ar_PowerFactor_L1: 				st_Variable:= IotExtractType(monitor.powermonitor.InternalSupply.ar_PowerFactor[1], 2, 0); 
// eDataMappingVarNames.powermonitor_InternalSupply_ar_PowerFactor_L2: 				st_Variable:= IotExtractType(monitor.powermonitor.InternalSupply.ar_PowerFactor[2], 2, 0); 
// eDataMappingVarNames.powermonitor_InternalSupply_ar_PowerFactor_L3: 				st_Variable:= IotExtractType(monitor.powermonitor.InternalSupply.ar_PowerFactor[3], 2, 0); 
// eDataMappingVarNames.powermonitor_InternalSupply_ar_Current_AVG: 				st_Variable:= IotExtractType(monitor.powermonitor.InternalSupply.ar_Current[0], 1, 1); 
// eDataMappingVarNames.powermonitor_InternalSupply_ar_Current_L1: 				st_Variable:= IotExtractType(monitor.powermonitor.InternalSupply.ar_Current[1], 1, 1); 
// eDataMappingVarNames.powermonitor_InternalSupply_ar_Current_L2: 				st_Variable:= IotExtractType(monitor.powermonitor.InternalSupply.ar_Current[2], 1, 1); 
// eDataMappingVarNames.powermonitor_InternalSupply_ar_Current_L3: 				st_Variable:= IotExtractType(monitor.powermonitor.InternalSupply.ar_Current[3], 1, 1); 
// eDataMappingVarNames.powermonitor_InternalSupply_ar_Current_N: 				st_Variable:= IotExtractType(monitor.powermonitor.InternalSupply.ar_Current[4]	  , 1, 1); 
// eDataMappingVarNames.powermonitor_InternalSupply_r_CurrentUnbalance: 				st_Variable:= IotExtractType(monitor.powermonitor.InternalSupply.r_CurrentUnbalance, 1, 0); 
// eDataMappingVarNames.powermonitor_BESS_e_ACrotationStatus: 				st_Variable:= IotExtractType(monitor.powermonitor.BESS.e_ACrotationStatus, 0, 0); 
// eDataMappingVarNames.powermonitor_BESS_ar_Current_AVG: 				st_Variable:= IotExtractType(monitor.powermonitor.BESS.ar_Current[0], 1, 1); 
// eDataMappingVarNames.powermonitor_BESS_ar_Current_L1: 				st_Variable:= IotExtractType(monitor.powermonitor.BESS.ar_Current[1], 1, 1); 
// eDataMappingVarNames.powermonitor_BESS_ar_Current_L2: 				st_Variable:= IotExtractType(monitor.powermonitor.BESS.ar_Current[2], 1, 1); 
// eDataMappingVarNames.powermonitor_BESS_ar_Current_L3: 				st_Variable:= IotExtractType(monitor.powermonitor.BESS.ar_Current[3], 1, 1); 
// eDataMappingVarNames.powermonitor_BESS_ar_Current_N: 				st_Variable:= IotExtractType(monitor.powermonitor.BESS.ar_Current[4], 1, 1); 
// eDataMappingVarNames.powermonitor_BESS_r_LineVoltage: 				st_Variable:= IotExtractType(monitor.powermonitor.BESS.r_LineVoltage, 1, 1); 
// eDataMappingVarNames.powermonitor_BESS_r_Frequency: 				st_Variable:= IotExtractType(monitor.powermonitor.BESS.r_Frequency, 2, 1); 
// eDataMappingVarNames.powermonitor_BESS_r_currentUnbalance: 				st_Variable:= IotExtractType(monitor.powermonitor.BESS.r_currentUnbalance, 1, 0); 
// eDataMappingVarNames.powermonitor_BESS_r_ApparentPower: 				st_Variable:= IotExtractType(monitor.powermonitor.BESS.r_ApparentPower	, 1, 1); 
// eDataMappingVarNames.powermonitor_BESS_r_ReactivePower: 				st_Variable:= IotExtractType(monitor.powermonitor.BESS.r_ReactivePower	, 1, 1); 
// eDataMappingVarNames.powermonitor_BESS_r_ActivePower: 				st_Variable:= IotExtractType(monitor.powermonitor.BESS.r_ActivePower		, 1, 1); 
// eDataMappingVarNames.powermonitor_BESS_r_EnergyConsumed: 				st_Variable:= IotExtractType(monitor.powermonitor.BESS.r_EnergyConsumed, 0, 0); 
// eDataMappingVarNames.powermonitor_BESS_r_EnergySupplied: 				st_Variable:= IotExtractType(monitor.powermonitor.BESS.r_EnergySupplied, 0, 0); 
// eDataMappingVarNames.powermonitor_BESS_r_PowerFactor: 				st_Variable:= IotExtractType(monitor.powermonitor.BESS.r_PowerFactor, 2, 0); 
// eDataMappingVarNames.powermonitor_events_b_MBCommWarning: 				st_Variable:= IotExtractType(monitor.powermonitor.events.b_MBCommWarning, 0, 0); 
// eDataMappingVarNames.powermonitor_events_b_MBCommError: 				st_Variable:= IotExtractType(monitor.powermonitor.events.b_MBCommError, 0, 0); 
// eDataMappingVarNames.powermonitor_events_b_MBTimeoutWarning: 				st_Variable:= IotExtractType(monitor.powermonitor.events.b_MBTimeoutWarning, 0, 0); 
// eDataMappingVarNames.powermonitor_events_b_EL3443Warning: 				st_Variable:= IotExtractType(monitor.powermonitor.events.b_EL3443Warning, 0, 0); 
// eDataMappingVarNames.powermonitor_events_b_EL3443Error: 				st_Variable:= IotExtractType(monitor.powermonitor.events.b_EL3443Error, 0, 0); 
// eDataMappingVarNames.powermonitor_events_b_ACdirectionDataInvalid: 				st_Variable:= IotExtractType(monitor.powermonitor.events.b_ACdirectionDataInvalid, 0, 0); 
// eDataMappingVarNames.ACswitchgear_b_InputSectionAvailable: 				st_Variable:= IotExtractType(monitor.ACswitchgear.b_InputSectionAvailable, 0, 0); 
// eDataMappingVarNames.ACswitchgear_b_InputMCCBfb: 				st_Variable:= IotExtractType(monitor.ACswitchgear.b_InputMCCBfb, 0, 0); 
// eDataMappingVarNames.ACswitchgear_b_InputMCCBShuntOK: 				st_Variable:= IotExtractType(monitor.ACswitchgear.b_InputMCCBShuntOK, 0, 0); 
// eDataMappingVarNames.ACswitchgear_b_OutputMCCBfb: 				st_Variable:= IotExtractType(monitor.ACswitchgear.b_OutputMCCBfb, 0, 0); 
// eDataMappingVarNames.ACswitchgear_b_OutputMCCBShuntOK: 				st_Variable:= IotExtractType(monitor.ACswitchgear.b_OutputMCCBShuntOK, 0, 0); 
// eDataMappingVarNames.ACswitchgear_b_CEEprefuseOK: 				st_Variable:= IotExtractType(monitor.ACswitchgear.b_CEEprefuseOK, 0, 0); 
// eDataMappingVarNames.ACswitchgear_b_InputSynchronizerfb: 				st_Variable:= IotExtractType(monitor.ACswitchgear.b_InputSynchronizerfb, 0, 0); 
// eDataMappingVarNames.ACswitchgear_b_InputContactorfb: 				st_Variable:= IotExtractType(monitor.ACswitchgear.b_InputContactorfb, 0, 0); 
// eDataMappingVarNames.ACswitchgear_b_PENlinkfb: 				st_Variable:= IotExtractType(monitor.ACswitchgear.b_PENlinkfb, 0, 0); 
// eDataMappingVarNames.ACswitchgear_events_b_InputMCCBShuntFault: 				st_Variable:= IotExtractType(monitor.ACswitchgear.events.b_InputMCCBShuntFault, 0, 0); 
// eDataMappingVarNames.ACswitchgear_events_b_OutputMCCBShuntFault: 				st_Variable:= IotExtractType(monitor.ACswitchgear.events.b_OutputMCCBShuntFault, 0, 0); 
// eDataMappingVarNames.ACswitchgear_events_b_CEEprefuseFault: 				st_Variable:= IotExtractType(monitor.ACswitchgear.events.b_CEEprefuseFault, 0, 0); 
// eDataMappingVarNames.ACswitchgear_events_b_InputContactorFault: 				st_Variable:= IotExtractType(monitor.ACswitchgear.events.b_InputContactorFault, 0, 0); 
// eDataMappingVarNames.neutraltransformer_b_active: 				st_Variable:= IotExtractType(monitor.neutraltransformer.b_active, 0, 0); 
// eDataMappingVarNames.neutraltransformer_r_TemperaturePhase_0: 				st_Variable:= IotExtractType(monitor.neutraltransformer.r_TemperaturePhase[0], 1, 0); 
// eDataMappingVarNames.neutraltransformer_r_TemperaturePhase_1: 				st_Variable:= IotExtractType(monitor.neutraltransformer.r_TemperaturePhase[1], 1, 0); 
// eDataMappingVarNames.neutraltransformer_r_TemperaturePhase_2: 				st_Variable:= IotExtractType(monitor.neutraltransformer.r_TemperaturePhase[2], 1, 0); 
// eDataMappingVarNames.neutraltransformer_r_TemperaturePhase_3: 				st_Variable:= IotExtractType(monitor.neutraltransformer.r_TemperaturePhase[3], 1, 0); 
// eDataMappingVarNames.neutraltransformer_r_TemperaturePhase_4: 				st_Variable:= IotExtractType(monitor.neutraltransformer.r_TemperaturePhase[4], 1, 0); 
// eDataMappingVarNames.neutraltransformer_r_TemperaturePhase_5: 				st_Variable:= IotExtractType(monitor.neutraltransformer.r_TemperaturePhase[5], 1, 0); 
// eDataMappingVarNames.neutraltransformer_r_TemperaturePhase_6: 				st_Variable:= IotExtractType(monitor.neutraltransformer.r_TemperaturePhase[6], 1, 0); 
// eDataMappingVarNames.neutraltransformer_r_Powerload: 				st_Variable:= IotExtractType(monitor.neutraltransformer.r_Powerload, 1, 0); 
// eDataMappingVarNames.neutraltransformer_r_ratedPower: 				st_Variable:= IotExtractType(monitor.neutraltransformer.r_ratedPower, 0, 0); 
// eDataMappingVarNames.neutraltransformer_events_b_TemperatureHighPhase_1: 				st_Variable:= IotExtractType(monitor.neutraltransformer.events.b_TemperatureHighPhase[1], 0, 0); 
// eDataMappingVarNames.neutraltransformer_events_b_TemperatureHighPhase_2: 				st_Variable:= IotExtractType(monitor.neutraltransformer.events.b_TemperatureHighPhase[2], 0, 0); 
// eDataMappingVarNames.neutraltransformer_events_b_TemperatureHighPhase_3: 				st_Variable:= IotExtractType(monitor.neutraltransformer.events.b_TemperatureHighPhase[3], 0, 0); 
// eDataMappingVarNames.neutraltransformer_events_b_TemperatureTooHighPhase_1: 				st_Variable:= IotExtractType(monitor.neutraltransformer.events.b_TemperatureTooHighPhase[1], 0, 0); 
// eDataMappingVarNames.neutraltransformer_events_b_TemperatureTooHighPhase_2: 				st_Variable:= IotExtractType(monitor.neutraltransformer.events.b_TemperatureTooHighPhase[2], 0, 0); 
// eDataMappingVarNames.neutraltransformer_events_b_TemperatureTooHighPhase_3: 				st_Variable:= IotExtractType(monitor.neutraltransformer.events.b_TemperatureTooHighPhase[3], 0, 0); 
// eDataMappingVarNames.neutraltransformer_events_b_VoltageUnbalanceHigh: 				st_Variable:= IotExtractType(monitor.neutraltransformer.events.b_VoltageUnbalanceHigh, 0, 0); 
// eDataMappingVarNames.neutraltransformer_events_b_VoltageUnbalanceTooHigh: 				st_Variable:= IotExtractType(monitor.neutraltransformer.events.b_VoltageUnbalanceTooHigh, 0, 0); 
// eDataMappingVarNames.neutraltransformer_events_b_NeutralCurrentHigh: 				st_Variable:= IotExtractType(monitor.neutraltransformer.events.b_NeutralCurrentHigh, 0, 0); 
// eDataMappingVarNames.neutraltransformer_events_b_NeutralCurrentTooHigh: 				st_Variable:= IotExtractType(monitor.neutraltransformer.events.b_NeutralCurrentTooHigh, 0, 0); 
// eDataMappingVarNames.neutraltransformer_events_b_OvercurrentWarning: 				st_Variable:= IotExtractType(monitor.neutraltransformer.events.b_OvercurrentWarning, 0, 0); 
// eDataMappingVarNames.neutraltransformer_events_b_OvercurrentAlarm: 				st_Variable:= IotExtractType(monitor.neutraltransformer.events.b_OvercurrentAlarm, 0, 0); 
// eDataMappingVarNames.DCswitchgear_b_CouplingState: 				st_Variable:= IotExtractType(monitor.DCswitchgear.b_CouplingState, 0, 0); 
// eDataMappingVarNames.DCswitchgear_r_Current: 				st_Variable:= IotExtractType(monitor.DCswitchgear.r_Current, 0, 0); 
// eDataMappingVarNames.DCswitchgear_r_ratedCurrent: 				st_Variable:= IotExtractType(monitor.DCswitchgear.r_ratedCurrent, 0, 0); 
// eDataMappingVarNames.battery_BatteryInfo_b_BMSHeartBeatOK: 				st_Variable:= IotExtractType(monitor.battery.BatteryInfo.b_BMSHeartBeatOK, 0, 0); 
// eDataMappingVarNames.battery_BatteryInfo_e_BMS_PowerOnStatus: 				st_Variable:= IotExtractType(monitor.battery.BatteryInfo.e_BMS_PowerOnStatus, 0, 0); 
// eDataMappingVarNames.battery_BatteryInfo_e_BMS_Status: 				st_Variable:= IotExtractType(monitor.battery.BatteryInfo.e_BMS_Status, 0, 0); 
// eDataMappingVarNames.battery_BatteryInfo_r_SystemVoltage: 				st_Variable:= IotExtractType(monitor.battery.BatteryInfo.r_SystemVoltage, 1, 0); 
// eDataMappingVarNames.battery_BatteryInfo_r_SystemCurrent: 				st_Variable:= IotExtractType(monitor.battery.BatteryInfo.r_SystemCurrent, 1, 0); 
// eDataMappingVarNames.battery_BatteryInfo_r_SOC: 				st_Variable:= IotExtractType(monitor.battery.BatteryInfo.r_SOC, 1, 0); 
// eDataMappingVarNames.battery_BatteryInfo_r_SOH: 				st_Variable:= IotExtractType(monitor.battery.BatteryInfo.r_SOH, 1, 0); 
// eDataMappingVarNames.battery_BatteryInfo_ar_CellVoltage_0: 				st_Variable:= IotExtractType(monitor.battery.BatteryInfo.ar_CellVoltage[0], 2, 0); 
// eDataMappingVarNames.battery_BatteryInfo_ar_CellVoltage_1: 				st_Variable:= IotExtractType(monitor.battery.BatteryInfo.ar_CellVoltage[1], 2, 0); 
// eDataMappingVarNames.battery_BatteryInfo_ar_CellVoltage_2: 				st_Variable:= IotExtractType(monitor.battery.BatteryInfo.ar_CellVoltage[2], 2, 0); 
// eDataMappingVarNames.battery_BatteryInfo_ar_CellTemperature_0: 				st_Variable:= IotExtractType(monitor.battery.BatteryInfo.ar_CellTemperature[0], 1, 0); 
// eDataMappingVarNames.battery_BatteryInfo_ar_CellTemperature_1: 				st_Variable:= IotExtractType(monitor.battery.BatteryInfo.ar_CellTemperature[1], 1, 0); 
// eDataMappingVarNames.battery_BatteryInfo_ar_CellTemperature_2: 				st_Variable:= IotExtractType(monitor.battery.BatteryInfo.ar_CellTemperature[2], 1, 0); 
// eDataMappingVarNames.battery_BatteryInfo_r_MaxChargeCurrentAllowed: 				st_Variable:= IotExtractType(monitor.battery.BatteryInfo.r_MaxChargeCurrentAllowed, 0, 0); 
// eDataMappingVarNames.battery_BatteryInfo_r_MaxDischargeCurrentAllowed: 				st_Variable:= IotExtractType(monitor.battery.BatteryInfo.r_MaxDischargeCurrentAllowed, 0, 0); 
// eDataMappingVarNames.battery_BatteryInfo_r_MaxChargePowerAllowed: 				st_Variable:= IotExtractType(monitor.battery.BatteryInfo.r_MaxChargePowerAllowed, 0, 0); 
// eDataMappingVarNames.battery_BatteryInfo_r_MaxDischargePowerAllowed: 				st_Variable:= IotExtractType(monitor.battery.BatteryInfo.r_MaxDischargePowerAllowed, 0, 0); 
// eDataMappingVarNames.battery_BatteryInfo_r_MaxSystemVoltageAllowed: 				st_Variable:= IotExtractType(monitor.battery.BatteryInfo.r_MaxSystemVoltageAllowed, 0, 0); 
// eDataMappingVarNames.battery_BatteryInfo_r_MinSystemVoltageAllowed: 				st_Variable:= IotExtractType(monitor.battery.BatteryInfo.r_MinSystemVoltageAllowed, 0, 0); 
// eDataMappingVarNames.battery_BatteryInfo_r_SystemPower: 				st_Variable:= IotExtractType(monitor.battery.BatteryInfo.r_SystemPower, 1, 0); 
// eDataMappingVarNames.battery_BatteryInfo_r_ChargeSOE: 				st_Variable:= IotExtractType(monitor.battery.BatteryInfo.r_ChargeSOE, 0, 0); 
// eDataMappingVarNames.battery_BatteryInfo_r_DischargeSOE: 				st_Variable:= IotExtractType(monitor.battery.BatteryInfo.r_DischargeSOE, 0, 0); 
// eDataMappingVarNames.battery_BatteryInfo_r_RemainingChargeEnergy: 				st_Variable:= IotExtractType(monitor.battery.BatteryInfo.r_RemainingChargeEnergy, 0, 0); 
// eDataMappingVarNames.battery_BatteryInfo_r_RemainingDischargeEnergy: 				st_Variable:= IotExtractType(monitor.battery.BatteryInfo.r_RemainingDischargeEnergy, 0, 0); 
// eDataMappingVarNames.battery_BatteryInfo_r_HistAccChargeEnergy: 				st_Variable:= IotExtractType(monitor.battery.BatteryInfo.r_HistAccChargeEnergy, 0, 0); 
// eDataMappingVarNames.battery_BatteryInfo_r_HistAccDischargeEnergy: 				st_Variable:= IotExtractType(monitor.battery.BatteryInfo.r_HistAccDischargeEnergy, 0, 0); 
// eDataMappingVarNames.battery_BatteryInfo_r_ratedPower: 				st_Variable:= IotExtractType(monitor.battery.BatteryInfo.r_ratedPower, 0, 0); 
// eDataMappingVarNames.battery_BatteryInfo_r_ratedCurrent: 				st_Variable:= IotExtractType(monitor.battery.BatteryInfo.r_ratedCurrent, 0, 0); 
// eDataMappingVarNames.battery_BatteryInfo_r_ratedEnergyCapacity: 				st_Variable:= IotExtractType(monitor.battery.BatteryInfo.r_ratedEnergyCapacity, 0, 0); 
// eDataMappingVarNames.battery_BatteryInfo_ui_CycleCount: 				st_Variable:= IotExtractType(monitor.battery.BatteryInfo.ui_CycleCount, 0, 0); 
// eDataMappingVarNames.battery_BatteryInfo_r_SOCScaled: 				st_Variable:= IotExtractType(monitor.battery.BatteryInfo.r_SOCScaled, 1, 0); 
// eDataMappingVarNames.battery_BatteryInfo_b_chargingAllowed: 				st_Variable:= IotExtractType(monitor.battery.BatteryInfo.b_chargingAllowed, 0, 0); 
// eDataMappingVarNames.battery_BatteryInfo_b_dischargingAllowed: 				st_Variable:= IotExtractType(monitor.battery.BatteryInfo.b_dischargingAllowed, 0, 0); 
// eDataMappingVarNames.battery_BatteryInfo_r_RemainingDischargeEnergyNett: 				st_Variable:= IotExtractType(monitor.battery.BatteryInfo.r_RemainingDischargeEnergyNett, 0, 0); 
// eDataMappingVarNames.battery_BatteryInfo_r_RemainingChargeEnergyNett: 				st_Variable:= IotExtractType(monitor.battery.BatteryInfo.r_RemainingChargeEnergyNett, 0, 0); 
// eDataMappingVarNames.battery_BatteryInfo_r_maxVoltageEver: 				st_Variable:= IotExtractType(monitor.battery.BatteryInfo.r_maxVoltageEver, 1, 0); 
// eDataMappingVarNames.battery_BatteryInfo_r_maxChargeCurrentEver: 				st_Variable:= IotExtractType(monitor.battery.BatteryInfo.r_maxChargeCurrentEver, 1, 0); 
// eDataMappingVarNames.battery_BatteryInfo_r_maxDischargeCurrentEver: 				st_Variable:= IotExtractType(monitor.battery.BatteryInfo.r_maxDischargeCurrentEver, 1, 0); 
// eDataMappingVarNames.battery_T_RemainingTimeToAutoCalibration: 				st_Variable:= IotExtractType(monitor.battery.T_RemainingTimeToAutoCalibration, 0, 0); 
// eDataMappingVarNames.battery_MBMU_GeneralSBMUStatus_0: 				st_Variable:= IotExtractType(monitor.battery.MBMU.GeneralSBMUStatus[0], 0, 0); 
// eDataMappingVarNames.battery_MBMU_GeneralSBMUStatus_1: 				st_Variable:= IotExtractType(monitor.battery.MBMU.GeneralSBMUStatus[1], 0, 0); 
// eDataMappingVarNames.battery_MBMU_GeneralSBMUStatus_2: 				st_Variable:= IotExtractType(monitor.battery.MBMU.GeneralSBMUStatus[2], 0, 0); 
// eDataMappingVarNames.battery_MBMU_GeneralSBMUStatus_3: 				st_Variable:= IotExtractType(monitor.battery.MBMU.GeneralSBMUStatus[3], 0, 0); 
// eDataMappingVarNames.battery_MBMU_GeneralSBMUStatus_4: 				st_Variable:= IotExtractType(monitor.battery.MBMU.GeneralSBMUStatus[4], 0, 0); 
// eDataMappingVarNames.battery_MBMU_GeneralSBMUStatus_5: 				st_Variable:= IotExtractType(monitor.battery.MBMU.GeneralSBMUStatus[5], 0, 0); 
// eDataMappingVarNames.battery_MBMU_GeneralSBMUStatus_6: 				st_Variable:= IotExtractType(monitor.battery.MBMU.GeneralSBMUStatus[6], 0, 0); 
// eDataMappingVarNames.battery_MBMU_GeneralSBMUStatus_7: 				st_Variable:= IotExtractType(monitor.battery.MBMU.GeneralSBMUStatus[7], 0, 0); 
// eDataMappingVarNames.battery_MBMU_GeneralSBMUStatus_8: 				st_Variable:= IotExtractType(monitor.battery.MBMU.GeneralSBMUStatus[8], 0, 0); 
// eDataMappingVarNames.battery_MBMU_GeneralSBMUStatus_9: 				st_Variable:= IotExtractType(monitor.battery.MBMU.GeneralSBMUStatus[9], 0, 0); 
// eDataMappingVarNames.battery_MBMU_GeneralSBMUStatus_10: 				st_Variable:= IotExtractType(monitor.battery.MBMU.GeneralSBMUStatus[10], 0, 0); 
// eDataMappingVarNames.battery_MBMU_GeneralSBMUStatus_11: 				st_Variable:= IotExtractType(monitor.battery.MBMU.GeneralSBMUStatus[11], 0, 0); 
// eDataMappingVarNames.battery_MBMU_GeneralSBMUStatus_12: 				st_Variable:= IotExtractType(monitor.battery.MBMU.GeneralSBMUStatus[12], 0, 0); 
// eDataMappingVarNames.battery_MBMU_GeneralSBMUStatus_13: 				st_Variable:= IotExtractType(monitor.battery.MBMU.GeneralSBMUStatus[13], 0, 0); 
// eDataMappingVarNames.battery_MBMU_GeneralSBMUStatus_14: 				st_Variable:= IotExtractType(monitor.battery.MBMU.GeneralSBMUStatus[14], 0, 0); 
// eDataMappingVarNames.battery_MBMU_GeneralSBMUStatus_15: 				st_Variable:= IotExtractType(monitor.battery.MBMU.GeneralSBMUStatus[15], 0, 0); 
// eDataMappingVarNames.battery_MBMU_MBMUStatus_0: 				st_Variable:= IotExtractType(monitor.battery.MBMU.MBMUStatus[0], 0, 0); 
// eDataMappingVarNames.battery_MBMU_MBMUStatus_1: 				st_Variable:= IotExtractType(monitor.battery.MBMU.MBMUStatus[1], 0, 0); 
// eDataMappingVarNames.battery_MBMU_MBMUStatus_2: 				st_Variable:= IotExtractType(monitor.battery.MBMU.MBMUStatus[2], 0, 0); 
// eDataMappingVarNames.battery_MBMU_MBMUStatus_3: 				st_Variable:= IotExtractType(monitor.battery.MBMU.MBMUStatus[3], 0, 0); 
// eDataMappingVarNames.battery_MBMU_MBMUStatus_4: 				st_Variable:= IotExtractType(monitor.battery.MBMU.MBMUStatus[4], 0, 0); 
// eDataMappingVarNames.battery_MBMU_MBMUStatus_5: 				st_Variable:= IotExtractType(monitor.battery.MBMU.MBMUStatus[5], 0, 0); 
// eDataMappingVarNames.battery_MBMU_MBMUStatus_6: 				st_Variable:= IotExtractType(monitor.battery.MBMU.MBMUStatus[6], 0, 0); 
// eDataMappingVarNames.battery_MBMU_MBMUStatus_7: 				st_Variable:= IotExtractType(monitor.battery.MBMU.MBMUStatus[7], 0, 0); 
// eDataMappingVarNames.battery_MBMU_MBMUStatus_8: 				st_Variable:= IotExtractType(monitor.battery.MBMU.MBMUStatus[8], 0, 0); 
// eDataMappingVarNames.battery_MBMU_MBMUStatus_9: 				st_Variable:= IotExtractType(monitor.battery.MBMU.MBMUStatus[9], 0, 0); 
// eDataMappingVarNames.battery_MBMU_MBMUStatus_10: 				st_Variable:= IotExtractType(monitor.battery.MBMU.MBMUStatus[10], 0, 0); 
// eDataMappingVarNames.battery_MBMU_MBMUStatus_11: 				st_Variable:= IotExtractType(monitor.battery.MBMU.MBMUStatus[11], 0, 0); 
// eDataMappingVarNames.battery_MBMU_MBMUStatus_12: 				st_Variable:= IotExtractType(monitor.battery.MBMU.MBMUStatus[12], 0, 0); 
// eDataMappingVarNames.battery_MBMU_MBMUStatus_13: 				st_Variable:= IotExtractType(monitor.battery.MBMU.MBMUStatus[13], 0, 0); 
// eDataMappingVarNames.battery_MBMU_MBMUStatus_14: 				st_Variable:= IotExtractType(monitor.battery.MBMU.MBMUStatus[14], 0, 0); 
// eDataMappingVarNames.battery_MBMU_MBMUStatus_15: 				st_Variable:= IotExtractType(monitor.battery.MBMU.MBMUStatus[15], 0, 0); 
// eDataMappingVarNames.battery_MBMU_s_MBMU_SWVer: 				st_Variable:= IotExtractType(monitor.battery.MBMU.s_MBMU_SWVer, 0, 0); 
// eDataMappingVarNames.battery_MBMU_s_MBMU_HWVer: 				st_Variable:= IotExtractType(monitor.battery.MBMU.s_MBMU_HWVer, 0, 0); 
// eDataMappingVarNames.battery_MBMU_s_ETH_SWVer: 				st_Variable:= IotExtractType(monitor.battery.MBMU.s_ETH_SWVer, 0, 0); 
// eDataMappingVarNames.battery_MBMU_r_ETH_HWVer: 				st_Variable:= IotExtractType(monitor.battery.MBMU.r_ETH_HWVer, 0, 0); 
// eDataMappingVarNames.battery_MBMU_by_NumberOfSubSystems: 				st_Variable:= IotExtractType(monitor.battery.MBMU.by_NumberOfSubSystems, 0, 0); 
// eDataMappingVarNames.battery_MBMU_DateTime_0: 				st_Variable:= IotExtractType(monitor.battery.MBMU.DateTime[0], 0, 0); 
// eDataMappingVarNames.battery_MBMU_DateTime_1: 				st_Variable:= IotExtractType(monitor.battery.MBMU.DateTime[1], 0, 0); 
// eDataMappingVarNames.battery_MBMU_DateTime_2: 				st_Variable:= IotExtractType(monitor.battery.MBMU.DateTime[2], 0, 0); 
// eDataMappingVarNames.battery_MBMU_DateTime_3: 				st_Variable:= IotExtractType(monitor.battery.MBMU.DateTime[3], 0, 0); 
// eDataMappingVarNames.battery_MBMU_DateTime_4: 				st_Variable:= IotExtractType(monitor.battery.MBMU.DateTime[4], 0, 0); 
// eDataMappingVarNames.battery_MBMU_DateTime_5: 				st_Variable:= IotExtractType(monitor.battery.MBMU.DateTime[5], 0, 0); 
// eDataMappingVarNames.battery_MBMU_b_InsulationSwitchOpen: 				st_Variable:= IotExtractType(monitor.battery.MBMU.b_InsulationSwitchOpen, 0, 0); 
// eDataMappingVarNames.battery_MBMU_BatteryStatus_b_BMSHeartBeatOK: 				st_Variable:= IotExtractType(monitor.battery.MBMU.BatteryStatus.b_BMSHeartBeatOK, 0, 0); 
// eDataMappingVarNames.battery_MBMU_BatteryStatus_e_BMS_PowerOnStatus: 				st_Variable:= IotExtractType(monitor.battery.MBMU.BatteryStatus.e_BMS_PowerOnStatus, 0, 0); 
// eDataMappingVarNames.battery_MBMU_BatteryStatus_e_BMS_Status: 					st_Variable:= IotExtractType(monitor.battery.MBMU.BatteryStatus.e_BMS_Status, 0, 0); 
// eDataMappingVarNames.battery_MBMU_BatteryStatus_r_SystemVoltage: 				st_Variable:= IotExtractType(monitor.battery.MBMU.BatteryStatus.r_SystemVoltage, 0, 0); 
// eDataMappingVarNames.battery_MBMU_BatteryStatus_r_SystemCurrent: 				st_Variable:= IotExtractType(monitor.battery.MBMU.BatteryStatus.r_SystemCurrent, 0, 0); 
// eDataMappingVarNames.battery_MBMU_BatteryStatus_r_SOC: 							st_Variable:= IotExtractType(monitor.battery.MBMU.BatteryStatus.r_SOC, 1, 0); 
// eDataMappingVarNames.battery_MBMU_BatteryStatus_r_SOH: 							st_Variable:= IotExtractType(monitor.battery.MBMU.BatteryStatus.r_SOH, 1, 0); 
// eDataMappingVarNames.battery_MBMU_BatteryStatus_ar_CellVoltage_0: 				st_Variable:= IotExtractType(monitor.battery.MBMU.BatteryStatus.ar_CellVoltage[0], 2, 0); 
// eDataMappingVarNames.battery_MBMU_BatteryStatus_ar_CellVoltage_1: 				st_Variable:= IotExtractType(monitor.battery.MBMU.BatteryStatus.ar_CellVoltage[1], 2, 0); 
// eDataMappingVarNames.battery_MBMU_BatteryStatus_ar_CellVoltage_2: 				st_Variable:= IotExtractType(monitor.battery.MBMU.BatteryStatus.ar_CellVoltage[2], 2, 0); 
// eDataMappingVarNames.battery_MBMU_BatteryStatus_ar_CellTemperature_0: 				st_Variable:= IotExtractType(monitor.battery.MBMU.BatteryStatus.ar_CellTemperature[0], 1, 0); 
// eDataMappingVarNames.battery_MBMU_BatteryStatus_ar_CellTemperature_1: 				st_Variable:= IotExtractType(monitor.battery.MBMU.BatteryStatus.ar_CellTemperature[1], 1, 0); 
// eDataMappingVarNames.battery_MBMU_BatteryStatus_ar_CellTemperature_2: 				st_Variable:= IotExtractType(monitor.battery.MBMU.BatteryStatus.ar_CellTemperature[2], 1, 0); 
// eDataMappingVarNames.battery_MBMU_BatteryStatus_r_MaxChargeCurrentAllowed: 				st_Variable:= IotExtractType(monitor.battery.MBMU.BatteryStatus.r_MaxChargeCurrentAllowed, 0, 0); 
// eDataMappingVarNames.battery_MBMU_BatteryStatus_r_MaxDischargeCurrentAllowed: 				st_Variable:= IotExtractType(monitor.battery.MBMU.BatteryStatus.r_MaxDischargeCurrentAllowed, 0, 0); 
// eDataMappingVarNames.battery_MBMU_BatteryStatus_r_MaxChargePowerAllowed: 				st_Variable:= IotExtractType(monitor.battery.MBMU.BatteryStatus.r_MaxChargePowerAllowed, 0, 0); 
// eDataMappingVarNames.battery_MBMU_BatteryStatus_r_MaxDischargePowerAllowed: 				st_Variable:= IotExtractType(monitor.battery.MBMU.BatteryStatus.r_MaxDischargePowerAllowed, 0, 0); 
// eDataMappingVarNames.battery_MBMU_BatteryStatus_r_MaxSystemVoltageAllowed: 				st_Variable:= IotExtractType(monitor.battery.MBMU.BatteryStatus.r_MaxSystemVoltageAllowed, 0, 0); 
// eDataMappingVarNames.battery_MBMU_BatteryStatus_r_MinSystemVoltageAllowed: 				st_Variable:= IotExtractType(monitor.battery.MBMU.BatteryStatus.r_MinSystemVoltageAllowed, 0, 0); 
// eDataMappingVarNames.battery_MBMU_BatteryStatus_r_SystemPower: 				st_Variable:= IotExtractType(monitor.battery.MBMU.BatteryStatus.r_SystemPower, 1, 0); 
// eDataMappingVarNames.battery_MBMU_BatteryStatus_r_ChargeSOE: 				st_Variable:= IotExtractType(monitor.battery.MBMU.BatteryStatus.r_ChargeSOE, 0, 0); 
// eDataMappingVarNames.battery_MBMU_BatteryStatus_r_DischargeSOE: 				st_Variable:= IotExtractType(monitor.battery.MBMU.BatteryStatus.r_DischargeSOE, 0, 0); 
// eDataMappingVarNames.battery_MBMU_BatteryStatus_r_RemainingChargeEnergy: 				st_Variable:= IotExtractType(monitor.battery.MBMU.BatteryStatus.r_RemainingChargeEnergy, 0, 0); 
// eDataMappingVarNames.battery_MBMU_BatteryStatus_r_RemainingDischargeEnergy: 				st_Variable:= IotExtractType(monitor.battery.MBMU.BatteryStatus.r_RemainingDischargeEnergy, 0, 0); 
// eDataMappingVarNames.battery_MBMU_BatteryStatus_r_HistAccChargeEnergy: 				st_Variable:= IotExtractType(monitor.battery.MBMU.BatteryStatus.r_HistAccChargeEnergy, 0, 0); 
// eDataMappingVarNames.battery_MBMU_BatteryStatus_r_HistAccDischargeEnergy: 				st_Variable:= IotExtractType(monitor.battery.MBMU.BatteryStatus.r_HistAccDischargeEnergy, 0, 0); 
// eDataMappingVarNames.battery_SBMU_0_w_SystemWarning: 				st_Variable:= IotExtractType(monitor.battery.SBMU[0].w_SystemWarning, 0, 0); 
// eDataMappingVarNames.battery_SBMU_1_w_SystemWarning: 				st_Variable:= IotExtractType(monitor.battery.SBMU[1].w_SystemWarning, 0, 0); 
// eDataMappingVarNames.battery_SBMU_2_w_SystemWarning: 				st_Variable:= IotExtractType(monitor.battery.SBMU[2].w_SystemWarning, 0, 0); 
// eDataMappingVarNames.battery_SBMU_3_w_SystemWarning: 				st_Variable:= IotExtractType(monitor.battery.SBMU[3].w_SystemWarning, 0, 0); 
// eDataMappingVarNames.battery_SBMU_0_SystemAlarm_0: 				st_Variable:= IotExtractType(monitor.battery.SBMU[0].SystemAlarm[0], 0, 0); 
// eDataMappingVarNames.battery_SBMU_1_SystemAlarm_0: 				st_Variable:= IotExtractType(monitor.battery.SBMU[1].SystemAlarm[0], 0, 0); 
// eDataMappingVarNames.battery_SBMU_2_SystemAlarm_0: 				st_Variable:= IotExtractType(monitor.battery.SBMU[2].SystemAlarm[0], 0, 0); 
// eDataMappingVarNames.battery_SBMU_3_SystemAlarm_0: 				st_Variable:= IotExtractType(monitor.battery.SBMU[3].SystemAlarm[0], 0, 0); 
// eDataMappingVarNames.battery_SBMU_0_SystemAlarm_1: 				st_Variable:= IotExtractType(monitor.battery.SBMU[0].SystemAlarm[1], 0, 0); 
// eDataMappingVarNames.battery_SBMU_1_SystemAlarm_1: 				st_Variable:= IotExtractType(monitor.battery.SBMU[1].SystemAlarm[1], 0, 0); 
// eDataMappingVarNames.battery_SBMU_2_SystemAlarm_1: 				st_Variable:= IotExtractType(monitor.battery.SBMU[2].SystemAlarm[1], 0, 0); 
// eDataMappingVarNames.battery_SBMU_3_SystemAlarm_1: 				st_Variable:= IotExtractType(monitor.battery.SBMU[3].SystemAlarm[1], 0, 0); 
// eDataMappingVarNames.battery_SBMU_0_SystemAlarm_2: 				st_Variable:= IotExtractType(monitor.battery.SBMU[0].SystemAlarm[2], 0, 0); 
// eDataMappingVarNames.battery_SBMU_1_SystemAlarm_2: 				st_Variable:= IotExtractType(monitor.battery.SBMU[1].SystemAlarm[2], 0, 0); 
// eDataMappingVarNames.battery_SBMU_2_SystemAlarm_2: 				st_Variable:= IotExtractType(monitor.battery.SBMU[2].SystemAlarm[2], 0, 0); 
// eDataMappingVarNames.battery_SBMU_3_SystemAlarm_2: 				st_Variable:= IotExtractType(monitor.battery.SBMU[3].SystemAlarm[2], 0, 0); 
// eDataMappingVarNames.battery_SBMU_0_b_PrechargeRelayClosed: 				st_Variable:= IotExtractType(monitor.battery.SBMU[0].b_PrechargeRelayClosed, 0, 0); 
// eDataMappingVarNames.battery_SBMU_1_b_PrechargeRelayClosed: 				st_Variable:= IotExtractType(monitor.battery.SBMU[1].b_PrechargeRelayClosed, 0, 0); 
// eDataMappingVarNames.battery_SBMU_2_b_PrechargeRelayClosed: 				st_Variable:= IotExtractType(monitor.battery.SBMU[2].b_PrechargeRelayClosed, 0, 0); 
// eDataMappingVarNames.battery_SBMU_3_b_PrechargeRelayClosed: 				st_Variable:= IotExtractType(monitor.battery.SBMU[3].b_PrechargeRelayClosed, 0, 0); 
// eDataMappingVarNames.battery_SBMU_0_b_MainPosRelayClosed: 				st_Variable:= IotExtractType(monitor.battery.SBMU[0].b_MainPosRelayClosed, 0, 0); 
// eDataMappingVarNames.battery_SBMU_1_b_MainPosRelayClosed: 				st_Variable:= IotExtractType(monitor.battery.SBMU[1].b_MainPosRelayClosed, 0, 0); 
// eDataMappingVarNames.battery_SBMU_2_b_MainPosRelayClosed: 				st_Variable:= IotExtractType(monitor.battery.SBMU[2].b_MainPosRelayClosed, 0, 0); 
// eDataMappingVarNames.battery_SBMU_3_b_MainPosRelayClosed: 				st_Variable:= IotExtractType(monitor.battery.SBMU[3].b_MainPosRelayClosed, 0, 0); 
// eDataMappingVarNames.battery_SBMU_0_b_MainNegRelayClosed: 				st_Variable:= IotExtractType(monitor.battery.SBMU[0].b_MainNegRelayClosed, 0, 0); 
// eDataMappingVarNames.battery_SBMU_1_b_MainNegRelayClosed: 				st_Variable:= IotExtractType(monitor.battery.SBMU[1].b_MainNegRelayClosed, 0, 0); 
// eDataMappingVarNames.battery_SBMU_2_b_MainNegRelayClosed: 				st_Variable:= IotExtractType(monitor.battery.SBMU[2].b_MainNegRelayClosed, 0, 0); 
// eDataMappingVarNames.battery_SBMU_3_b_MainNegRelayClosed: 				st_Variable:= IotExtractType(monitor.battery.SBMU[3].b_MainNegRelayClosed, 0, 0); 
// eDataMappingVarNames.battery_SBMU_0_b_ControlBoxFanOn: 				st_Variable:= IotExtractType(monitor.battery.SBMU[0].b_ControlBoxFanOn, 0, 0); 
// eDataMappingVarNames.battery_SBMU_1_b_ControlBoxFanOn: 				st_Variable:= IotExtractType(monitor.battery.SBMU[1].b_ControlBoxFanOn, 0, 0); 
// eDataMappingVarNames.battery_SBMU_2_b_ControlBoxFanOn: 				st_Variable:= IotExtractType(monitor.battery.SBMU[2].b_ControlBoxFanOn, 0, 0); 
// eDataMappingVarNames.battery_SBMU_3_b_ControlBoxFanOn: 				st_Variable:= IotExtractType(monitor.battery.SBMU[3].b_ControlBoxFanOn, 0, 0); 
// eDataMappingVarNames.battery_SBMU_0_b_BalanceStatus: 				st_Variable:= IotExtractType(monitor.battery.SBMU[0].b_BalanceStatus, 0, 0); 
// eDataMappingVarNames.battery_SBMU_1_b_BalanceStatus: 				st_Variable:= IotExtractType(monitor.battery.SBMU[1].b_BalanceStatus, 0, 0); 
// eDataMappingVarNames.battery_SBMU_2_b_BalanceStatus: 				st_Variable:= IotExtractType(monitor.battery.SBMU[2].b_BalanceStatus, 0, 0); 
// eDataMappingVarNames.battery_SBMU_3_b_BalanceStatus: 				st_Variable:= IotExtractType(monitor.battery.SBMU[3].b_BalanceStatus, 0, 0); 
// eDataMappingVarNames.battery_SBMU_0_b_DoorState: 				st_Variable:= IotExtractType(monitor.battery.SBMU[0].b_DoorState, 0, 0); 
// eDataMappingVarNames.battery_SBMU_1_b_DoorState: 				st_Variable:= IotExtractType(monitor.battery.SBMU[1].b_DoorState, 0, 0); 
// eDataMappingVarNames.battery_SBMU_2_b_DoorState: 				st_Variable:= IotExtractType(monitor.battery.SBMU[2].b_DoorState, 0, 0); 
// eDataMappingVarNames.battery_SBMU_3_b_DoorState: 				st_Variable:= IotExtractType(monitor.battery.SBMU[3].b_DoorState, 0, 0); 
// eDataMappingVarNames.battery_SBMU_0_s_SBMU_SWVer: 				st_Variable:= IotExtractType(monitor.battery.SBMU[0].s_SBMU_SWVer, 0, 0); 
// eDataMappingVarNames.battery_SBMU_1_s_SBMU_SWVer: 				st_Variable:= IotExtractType(monitor.battery.SBMU[1].s_SBMU_SWVer, 0, 0); 
// eDataMappingVarNames.battery_SBMU_2_s_SBMU_SWVer: 				st_Variable:= IotExtractType(monitor.battery.SBMU[2].s_SBMU_SWVer, 0, 0); 
// eDataMappingVarNames.battery_SBMU_3_s_SBMU_SWVer: 				st_Variable:= IotExtractType(monitor.battery.SBMU[3].s_SBMU_SWVer, 0, 0); 
// eDataMappingVarNames.battery_SBMU_0_s_SBMU_HWVer: 				st_Variable:= IotExtractType(monitor.battery.SBMU[0].s_SBMU_HWVer, 0, 0); 
// eDataMappingVarNames.battery_SBMU_1_s_SBMU_HWVer: 				st_Variable:= IotExtractType(monitor.battery.SBMU[1].s_SBMU_HWVer, 0, 0); 
// eDataMappingVarNames.battery_SBMU_2_s_SBMU_HWVer: 				st_Variable:= IotExtractType(monitor.battery.SBMU[2].s_SBMU_HWVer, 0, 0); 
// eDataMappingVarNames.battery_SBMU_3_s_SBMU_HWVer: 				st_Variable:= IotExtractType(monitor.battery.SBMU[3].s_SBMU_HWVer, 0, 0); 
// eDataMappingVarNames.battery_SBMU_0_s_CSC_SWVer: 				st_Variable:= IotExtractType(monitor.battery.SBMU[0].s_CSC_SWVer, 0, 0); 
// eDataMappingVarNames.battery_SBMU_1_s_CSC_SWVer: 				st_Variable:= IotExtractType(monitor.battery.SBMU[1].s_CSC_SWVer, 0, 0); 
// eDataMappingVarNames.battery_SBMU_2_s_CSC_SWVer: 				st_Variable:= IotExtractType(monitor.battery.SBMU[2].s_CSC_SWVer, 0, 0); 
// eDataMappingVarNames.battery_SBMU_3_s_CSC_SWVer: 				st_Variable:= IotExtractType(monitor.battery.SBMU[3].s_CSC_SWVer, 0, 0); 
// eDataMappingVarNames.battery_SBMU_0_s_CSC_HWVer: 				st_Variable:= IotExtractType(monitor.battery.SBMU[0].s_CSC_HWVer, 0, 0); 
// eDataMappingVarNames.battery_SBMU_1_s_CSC_HWVer: 				st_Variable:= IotExtractType(monitor.battery.SBMU[1].s_CSC_HWVer, 0, 0); 
// eDataMappingVarNames.battery_SBMU_2_s_CSC_HWVer: 				st_Variable:= IotExtractType(monitor.battery.SBMU[2].s_CSC_HWVer, 0, 0); 
// eDataMappingVarNames.battery_SBMU_3_s_CSC_HWVer: 				st_Variable:= IotExtractType(monitor.battery.SBMU[3].s_CSC_HWVer, 0, 0); 
// eDataMappingVarNames.battery_SBMU_0_BatteryStatus_r_SystemVoltage: 				st_Variable:= IotExtractType(monitor.battery.SBMU[0].BatteryStatus.r_SystemVoltage, 1, 0); 
// eDataMappingVarNames.battery_SBMU_1_BatteryStatus_r_SystemVoltage: 				st_Variable:= IotExtractType(monitor.battery.SBMU[1].BatteryStatus.r_SystemVoltage, 1, 0); 
// eDataMappingVarNames.battery_SBMU_2_BatteryStatus_r_SystemVoltage: 				st_Variable:= IotExtractType(monitor.battery.SBMU[2].BatteryStatus.r_SystemVoltage, 1, 0); 
// eDataMappingVarNames.battery_SBMU_3_BatteryStatus_r_SystemVoltage: 				st_Variable:= IotExtractType(monitor.battery.SBMU[3].BatteryStatus.r_SystemVoltage, 1, 0); 
// eDataMappingVarNames.battery_SBMU_0_BatteryStatus_r_SystemCurrent: 				st_Variable:= IotExtractType(monitor.battery.SBMU[0].BatteryStatus.r_SystemCurrent, 1, 0); 
// eDataMappingVarNames.battery_SBMU_1_BatteryStatus_r_SystemCurrent: 				st_Variable:= IotExtractType(monitor.battery.SBMU[1].BatteryStatus.r_SystemCurrent, 1, 0); 
// eDataMappingVarNames.battery_SBMU_2_BatteryStatus_r_SystemCurrent: 				st_Variable:= IotExtractType(monitor.battery.SBMU[2].BatteryStatus.r_SystemCurrent, 1, 0); 
// eDataMappingVarNames.battery_SBMU_3_BatteryStatus_r_SystemCurrent: 				st_Variable:= IotExtractType(monitor.battery.SBMU[3].BatteryStatus.r_SystemCurrent, 1, 0); 
// eDataMappingVarNames.battery_SBMU_0_BatteryStatus_r_SOC: 				st_Variable:= IotExtractType(monitor.battery.SBMU[0].BatteryStatus.r_SOC, 1, 0); 
// eDataMappingVarNames.battery_SBMU_1_BatteryStatus_r_SOC: 				st_Variable:= IotExtractType(monitor.battery.SBMU[1].BatteryStatus.r_SOC, 1, 0); 
// eDataMappingVarNames.battery_SBMU_2_BatteryStatus_r_SOC: 				st_Variable:= IotExtractType(monitor.battery.SBMU[2].BatteryStatus.r_SOC, 1, 0); 
// eDataMappingVarNames.battery_SBMU_3_BatteryStatus_r_SOC: 				st_Variable:= IotExtractType(monitor.battery.SBMU[3].BatteryStatus.r_SOC, 1, 0); 
// eDataMappingVarNames.battery_SBMU_0_BatteryStatus_r_SOH: 				st_Variable:= IotExtractType(monitor.battery.SBMU[0].BatteryStatus.r_SOH, 1, 0); 
// eDataMappingVarNames.battery_SBMU_1_BatteryStatus_r_SOH: 				st_Variable:= IotExtractType(monitor.battery.SBMU[1].BatteryStatus.r_SOH, 1, 0); 
// eDataMappingVarNames.battery_SBMU_2_BatteryStatus_r_SOH: 				st_Variable:= IotExtractType(monitor.battery.SBMU[2].BatteryStatus.r_SOH, 1, 0); 
// eDataMappingVarNames.battery_SBMU_3_BatteryStatus_r_SOH: 				st_Variable:= IotExtractType(monitor.battery.SBMU[3].BatteryStatus.r_SOH, 1, 0); 
// eDataMappingVarNames.battery_SBMU_0_BatteryStatus_ar_CellVoltage_0: 				st_Variable:= IotExtractType(monitor.battery.SBMU[0].BatteryStatus.ar_CellVoltage[0], 2, 0); 
// eDataMappingVarNames.battery_SBMU_1_BatteryStatus_ar_CellVoltage_0: 				st_Variable:= IotExtractType(monitor.battery.SBMU[1].BatteryStatus.ar_CellVoltage[0], 2, 0); 
// eDataMappingVarNames.battery_SBMU_2_BatteryStatus_ar_CellVoltage_0: 				st_Variable:= IotExtractType(monitor.battery.SBMU[2].BatteryStatus.ar_CellVoltage[0], 2, 0); 
// eDataMappingVarNames.battery_SBMU_3_BatteryStatus_ar_CellVoltage_0: 				st_Variable:= IotExtractType(monitor.battery.SBMU[3].BatteryStatus.ar_CellVoltage[0], 2, 0); 
// eDataMappingVarNames.battery_SBMU_0_BatteryStatus_ar_CellVoltage_1: 				st_Variable:= IotExtractType(monitor.battery.SBMU[0].BatteryStatus.ar_CellVoltage[1], 2, 0); 
// eDataMappingVarNames.battery_SBMU_1_BatteryStatus_ar_CellVoltage_1: 				st_Variable:= IotExtractType(monitor.battery.SBMU[1].BatteryStatus.ar_CellVoltage[1], 2, 0); 
// eDataMappingVarNames.battery_SBMU_2_BatteryStatus_ar_CellVoltage_1: 				st_Variable:= IotExtractType(monitor.battery.SBMU[2].BatteryStatus.ar_CellVoltage[1], 2, 0); 
// eDataMappingVarNames.battery_SBMU_3_BatteryStatus_ar_CellVoltage_1: 				st_Variable:= IotExtractType(monitor.battery.SBMU[3].BatteryStatus.ar_CellVoltage[1], 2, 0); 
// eDataMappingVarNames.battery_SBMU_0_BatteryStatus_ar_CellVoltage_2: 				st_Variable:= IotExtractType(monitor.battery.SBMU[0].BatteryStatus.ar_CellVoltage[2], 2, 0); 
// eDataMappingVarNames.battery_SBMU_1_BatteryStatus_ar_CellVoltage_2: 				st_Variable:= IotExtractType(monitor.battery.SBMU[1].BatteryStatus.ar_CellVoltage[2], 2, 0); 
// eDataMappingVarNames.battery_SBMU_2_BatteryStatus_ar_CellVoltage_2: 				st_Variable:= IotExtractType(monitor.battery.SBMU[2].BatteryStatus.ar_CellVoltage[2], 2, 0); 
// eDataMappingVarNames.battery_SBMU_3_BatteryStatus_ar_CellVoltage_2: 				st_Variable:= IotExtractType(monitor.battery.SBMU[3].BatteryStatus.ar_CellVoltage[2], 2, 0); 
// eDataMappingVarNames.battery_SBMU_0_BatteryStatus_ar_CellTemperature_0: 				st_Variable:= IotExtractType(monitor.battery.SBMU[0].BatteryStatus.ar_CellTemperature[0], 1, 0); 
// eDataMappingVarNames.battery_SBMU_1_BatteryStatus_ar_CellTemperature_0: 				st_Variable:= IotExtractType(monitor.battery.SBMU[1].BatteryStatus.ar_CellTemperature[0], 1, 0); 
// eDataMappingVarNames.battery_SBMU_2_BatteryStatus_ar_CellTemperature_0: 				st_Variable:= IotExtractType(monitor.battery.SBMU[2].BatteryStatus.ar_CellTemperature[0], 1, 0); 
// eDataMappingVarNames.battery_SBMU_3_BatteryStatus_ar_CellTemperature_0: 				st_Variable:= IotExtractType(monitor.battery.SBMU[3].BatteryStatus.ar_CellTemperature[0], 1, 0); 
// eDataMappingVarNames.battery_SBMU_0_BatteryStatus_ar_CellTemperature_1: 				st_Variable:= IotExtractType(monitor.battery.SBMU[0].BatteryStatus.ar_CellTemperature[1], 1, 0); 
// eDataMappingVarNames.battery_SBMU_1_BatteryStatus_ar_CellTemperature_1: 				st_Variable:= IotExtractType(monitor.battery.SBMU[1].BatteryStatus.ar_CellTemperature[1], 1, 0); 
// eDataMappingVarNames.battery_SBMU_2_BatteryStatus_ar_CellTemperature_1: 				st_Variable:= IotExtractType(monitor.battery.SBMU[2].BatteryStatus.ar_CellTemperature[1], 1, 0); 
// eDataMappingVarNames.battery_SBMU_3_BatteryStatus_ar_CellTemperature_1: 				st_Variable:= IotExtractType(monitor.battery.SBMU[3].BatteryStatus.ar_CellTemperature[1], 1, 0); 
// eDataMappingVarNames.battery_SBMU_0_BatteryStatus_ar_CellTemperature_2: 				st_Variable:= IotExtractType(monitor.battery.SBMU[0].BatteryStatus.ar_CellTemperature[2], 1, 0); 
// eDataMappingVarNames.battery_SBMU_1_BatteryStatus_ar_CellTemperature_2: 				st_Variable:= IotExtractType(monitor.battery.SBMU[1].BatteryStatus.ar_CellTemperature[2], 1, 0); 
// eDataMappingVarNames.battery_SBMU_2_BatteryStatus_ar_CellTemperature_2: 				st_Variable:= IotExtractType(monitor.battery.SBMU[2].BatteryStatus.ar_CellTemperature[2], 1, 0); 
// eDataMappingVarNames.battery_SBMU_3_BatteryStatus_ar_CellTemperature_2: 				st_Variable:= IotExtractType(monitor.battery.SBMU[3].BatteryStatus.ar_CellTemperature[2], 1, 0); 
// eDataMappingVarNames.battery_SBMU_0_BatteryStatus_r_MaxChargeCurrentAllowed: 				st_Variable:= IotExtractType(monitor.battery.SBMU[0].BatteryStatus.r_MaxChargeCurrentAllowed, 0, 0); 
// eDataMappingVarNames.battery_SBMU_1_BatteryStatus_r_MaxChargeCurrentAllowed: 				st_Variable:= IotExtractType(monitor.battery.SBMU[1].BatteryStatus.r_MaxChargeCurrentAllowed, 0, 0); 
// eDataMappingVarNames.battery_SBMU_2_BatteryStatus_r_MaxChargeCurrentAllowed: 				st_Variable:= IotExtractType(monitor.battery.SBMU[2].BatteryStatus.r_MaxChargeCurrentAllowed, 0, 0); 
// eDataMappingVarNames.battery_SBMU_3_BatteryStatus_r_MaxChargeCurrentAllowed: 				st_Variable:= IotExtractType(monitor.battery.SBMU[3].BatteryStatus.r_MaxChargeCurrentAllowed, 0, 0); 
// eDataMappingVarNames.battery_SBMU_0_BatteryStatus_r_MaxDischargeCurrentAllowed: 				st_Variable:= IotExtractType(monitor.battery.SBMU[0].BatteryStatus.r_MaxDischargeCurrentAllowed, 0, 0); 
// eDataMappingVarNames.battery_SBMU_1_BatteryStatus_r_MaxDischargeCurrentAllowed: 				st_Variable:= IotExtractType(monitor.battery.SBMU[1].BatteryStatus.r_MaxDischargeCurrentAllowed, 0, 0); 
// eDataMappingVarNames.battery_SBMU_2_BatteryStatus_r_MaxDischargeCurrentAllowed: 				st_Variable:= IotExtractType(monitor.battery.SBMU[2].BatteryStatus.r_MaxDischargeCurrentAllowed, 0, 0); 
// eDataMappingVarNames.battery_SBMU_3_BatteryStatus_r_MaxDischargeCurrentAllowed: 				st_Variable:= IotExtractType(monitor.battery.SBMU[3].BatteryStatus.r_MaxDischargeCurrentAllowed, 0, 0); 
// eDataMappingVarNames.battery_SBMU_0_BatteryStatus_r_HistAccChargeEnergy: 				st_Variable:= IotExtractType(monitor.battery.SBMU[0].BatteryStatus.r_HistAccChargeEnergy, 0, 0); 
// eDataMappingVarNames.battery_SBMU_1_BatteryStatus_r_HistAccChargeEnergy: 				st_Variable:= IotExtractType(monitor.battery.SBMU[1].BatteryStatus.r_HistAccChargeEnergy, 0, 0); 
// eDataMappingVarNames.battery_SBMU_2_BatteryStatus_r_HistAccChargeEnergy: 				st_Variable:= IotExtractType(monitor.battery.SBMU[2].BatteryStatus.r_HistAccChargeEnergy, 0, 0); 
// eDataMappingVarNames.battery_SBMU_3_BatteryStatus_r_HistAccChargeEnergy: 				st_Variable:= IotExtractType(monitor.battery.SBMU[3].BatteryStatus.r_HistAccChargeEnergy, 0, 0); 
// eDataMappingVarNames.battery_SBMU_0_BatteryStatus_r_HistAccDischargeEnergy: 				st_Variable:= IotExtractType(monitor.battery.SBMU[0].BatteryStatus.r_HistAccDischargeEnergy, 0, 0); 
// eDataMappingVarNames.battery_SBMU_1_BatteryStatus_r_HistAccDischargeEnergy: 				st_Variable:= IotExtractType(monitor.battery.SBMU[1].BatteryStatus.r_HistAccDischargeEnergy, 0, 0); 
// eDataMappingVarNames.battery_SBMU_2_BatteryStatus_r_HistAccDischargeEnergy: 				st_Variable:= IotExtractType(monitor.battery.SBMU[2].BatteryStatus.r_HistAccDischargeEnergy, 0, 0); 
// eDataMappingVarNames.battery_SBMU_3_BatteryStatus_r_HistAccDischargeEnergy: 				st_Variable:= IotExtractType(monitor.battery.SBMU[3].BatteryStatus.r_HistAccDischargeEnergy, 0, 0); 
// eDataMappingVarNames.battery_SBMU_0_BatteryStatus_w_MaxVoltageCellLocation: 				st_Variable:= IotExtractType(monitor.battery.SBMU[0].BatteryStatus.w_MaxVoltageCellLocation, 0, 0); 
// eDataMappingVarNames.battery_SBMU_1_BatteryStatus_w_MaxVoltageCellLocation: 				st_Variable:= IotExtractType(monitor.battery.SBMU[1].BatteryStatus.w_MaxVoltageCellLocation, 0, 0); 
// eDataMappingVarNames.battery_SBMU_2_BatteryStatus_w_MaxVoltageCellLocation: 				st_Variable:= IotExtractType(monitor.battery.SBMU[2].BatteryStatus.w_MaxVoltageCellLocation, 0, 0); 
// eDataMappingVarNames.battery_SBMU_3_BatteryStatus_w_MaxVoltageCellLocation: 				st_Variable:= IotExtractType(monitor.battery.SBMU[3].BatteryStatus.w_MaxVoltageCellLocation, 0, 0); 
// eDataMappingVarNames.battery_SBMU_0_BatteryStatus_w_MinVoltageCellLocation: 				st_Variable:= IotExtractType(monitor.battery.SBMU[0].BatteryStatus.w_MinVoltageCellLocation, 0, 0); 
// eDataMappingVarNames.battery_SBMU_1_BatteryStatus_w_MinVoltageCellLocation: 				st_Variable:= IotExtractType(monitor.battery.SBMU[1].BatteryStatus.w_MinVoltageCellLocation, 0, 0); 
// eDataMappingVarNames.battery_SBMU_2_BatteryStatus_w_MinVoltageCellLocation: 				st_Variable:= IotExtractType(monitor.battery.SBMU[2].BatteryStatus.w_MinVoltageCellLocation, 0, 0); 
// eDataMappingVarNames.battery_SBMU_3_BatteryStatus_w_MinVoltageCellLocation: 				st_Variable:= IotExtractType(monitor.battery.SBMU[3].BatteryStatus.w_MinVoltageCellLocation, 0, 0); 
// eDataMappingVarNames.battery_SBMU_0_BatteryStatus_w_MaxTempCellLocation: 				st_Variable:= IotExtractType(monitor.battery.SBMU[0].BatteryStatus.w_MaxTempCellLocation, 0, 0); 
// eDataMappingVarNames.battery_SBMU_1_BatteryStatus_w_MaxTempCellLocation: 				st_Variable:= IotExtractType(monitor.battery.SBMU[1].BatteryStatus.w_MaxTempCellLocation, 0, 0); 
// eDataMappingVarNames.battery_SBMU_2_BatteryStatus_w_MaxTempCellLocation: 				st_Variable:= IotExtractType(monitor.battery.SBMU[2].BatteryStatus.w_MaxTempCellLocation, 0, 0); 
// eDataMappingVarNames.battery_SBMU_3_BatteryStatus_w_MaxTempCellLocation: 				st_Variable:= IotExtractType(monitor.battery.SBMU[3].BatteryStatus.w_MaxTempCellLocation, 0, 0); 
// eDataMappingVarNames.battery_SBMU_0_BatteryStatus_w_MinTempCellLocation: 				st_Variable:= IotExtractType(monitor.battery.SBMU[0].BatteryStatus.w_MinTempCellLocation, 0, 0); 
// eDataMappingVarNames.battery_SBMU_1_BatteryStatus_w_MinTempCellLocation: 				st_Variable:= IotExtractType(monitor.battery.SBMU[1].BatteryStatus.w_MinTempCellLocation, 0, 0); 
// eDataMappingVarNames.battery_SBMU_2_BatteryStatus_w_MinTempCellLocation: 				st_Variable:= IotExtractType(monitor.battery.SBMU[2].BatteryStatus.w_MinTempCellLocation, 0, 0); 
// eDataMappingVarNames.battery_SBMU_3_BatteryStatus_w_MinTempCellLocation: 				st_Variable:= IotExtractType(monitor.battery.SBMU[3].BatteryStatus.w_MinTempCellLocation, 0, 0); 
// eDataMappingVarNames.battery_Events_b_COMMUNICATION_ERROR: 				st_Variable:= IotExtractType(monitor.battery.Events.b_COMMUNICATION_ERROR, 0, 0); 
// eDataMappingVarNames.battery_Events_b_OVER_TEMP_ALARM: 				st_Variable:= IotExtractType(monitor.battery.Events.b_OVER_TEMP_ALARM, 0, 0); 
// eDataMappingVarNames.battery_Events_b_OVER_TEMP_WARNING: 				st_Variable:= IotExtractType(monitor.battery.Events.b_OVER_TEMP_WARNING, 0, 0); 
// eDataMappingVarNames.battery_Events_b_UNDER_TEMP_ALARM: 				st_Variable:= IotExtractType(monitor.battery.Events.b_UNDER_TEMP_ALARM, 0, 0); 
// eDataMappingVarNames.battery_Events_b_UNDER_TEMP_WARNING: 				st_Variable:= IotExtractType(monitor.battery.Events.b_UNDER_TEMP_WARNING, 0, 0); 
// eDataMappingVarNames.battery_Events_b_OVER_CHARGE_CURRENT_ALARM: 				st_Variable:= IotExtractType(monitor.battery.Events.b_OVER_CHARGE_CURRENT_ALARM, 0, 0); 
// eDataMappingVarNames.battery_Events_b_OVER_CHARGE_CURRENT_WARNING: 				st_Variable:= IotExtractType(monitor.battery.Events.b_OVER_CHARGE_CURRENT_WARNING, 0, 0); 
// eDataMappingVarNames.battery_Events_b_OVER_DISCHARGE_CURRENT_ALARM: 				st_Variable:= IotExtractType(monitor.battery.Events.b_OVER_DISCHARGE_CURRENT_ALARM, 0, 0); 
// eDataMappingVarNames.battery_Events_b_OVER_DISCHARGE_CURRENT_WARNING: 				st_Variable:= IotExtractType(monitor.battery.Events.b_OVER_DISCHARGE_CURRENT_WARNING, 0, 0); 
// eDataMappingVarNames.battery_Events_b_OVER_VOLT_ALARM: 				st_Variable:= IotExtractType(monitor.battery.Events.b_OVER_VOLT_ALARM, 0, 0); 
// eDataMappingVarNames.battery_Events_b_OVER_VOLT_WARNING: 				st_Variable:= IotExtractType(monitor.battery.Events.b_OVER_VOLT_WARNING, 0, 0); 
// eDataMappingVarNames.battery_Events_b_UNDER_VOLT_ALARM: 				st_Variable:= IotExtractType(monitor.battery.Events.b_UNDER_VOLT_ALARM, 0, 0); 
// eDataMappingVarNames.battery_Events_b_UNDER_VOLT_WARNING: 				st_Variable:= IotExtractType(monitor.battery.Events.b_UNDER_VOLT_WARNING, 0, 0); 
// eDataMappingVarNames.battery_Events_b_UNDER_SOC_MIN_ALARM: 				st_Variable:= IotExtractType(monitor.battery.Events.b_UNDER_SOC_MIN_ALARM, 0, 0); 
// eDataMappingVarNames.battery_Events_b_UNDER_SOC_MIN_WARNING: 				st_Variable:= IotExtractType(monitor.battery.Events.b_UNDER_SOC_MIN_WARNING, 0, 0); 
// eDataMappingVarNames.battery_Events_b_OVER_SOC_MAX_ALARM: 				st_Variable:= IotExtractType(monitor.battery.Events.b_OVER_SOC_MAX_ALARM, 0, 0); 
// eDataMappingVarNames.battery_Events_b_OVER_SOC_MAX_WARNING: 				st_Variable:= IotExtractType(monitor.battery.Events.b_OVER_SOC_MAX_WARNING, 0, 0); 
// eDataMappingVarNames.battery_Events_b_VOLTAGE_IMBALANCE_WARNING: 				st_Variable:= IotExtractType(monitor.battery.Events.b_VOLTAGE_IMBALANCE_WARNING, 0, 0); 
// eDataMappingVarNames.battery_Events_b_TEMPERATURE_IMBALANCE_ALARM: 				st_Variable:= IotExtractType(monitor.battery.Events.b_TEMPERATURE_IMBALANCE_ALARM, 0, 0); 
// eDataMappingVarNames.battery_Events_b_TEMPERATURE_IMBALANCE_WARNING: 				st_Variable:= IotExtractType(monitor.battery.Events.b_TEMPERATURE_IMBALANCE_WARNING, 0, 0); 
// eDataMappingVarNames.battery_Events_b_CONTACTOR_ERROR: 				st_Variable:= IotExtractType(monitor.battery.Events.b_CONTACTOR_ERROR, 0, 0); 
// eDataMappingVarNames.battery_Events_b_FAN_ERROR: 				st_Variable:= IotExtractType(monitor.battery.Events.b_FAN_ERROR, 0, 0); 
// eDataMappingVarNames.battery_Events_b_GROUND_FAULT: 				st_Variable:= IotExtractType(monitor.battery.Events.b_GROUND_FAULT, 0, 0); 
// eDataMappingVarNames.battery_Events_b_OPEN_DOOR_ERROR: 				st_Variable:= IotExtractType(monitor.battery.Events.b_OPEN_DOOR_ERROR, 0, 0); 
// eDataMappingVarNames.battery_Events_b_CURRENT_IMBALANCE_WARNING: 				st_Variable:= IotExtractType(monitor.battery.Events.b_CURRENT_IMBALANCE_WARNING, 0, 0); 
// eDataMappingVarNames.battery_Events_b_OTHER_ALARM: 				st_Variable:= IotExtractType(monitor.battery.Events.b_OTHER_ALARM, 0, 0); 
// eDataMappingVarNames.battery_Events_b_OTHER_WARNING: 				st_Variable:= IotExtractType(monitor.battery.Events.b_OTHER_WARNING, 0, 0); 
// eDataMappingVarNames.battery_Events_b_CONFIGURATION_ALARM: 				st_Variable:= IotExtractType(monitor.battery.Events.b_CONFIGURATION_ALARM, 0, 0); 
// eDataMappingVarNames.battery_Events_b_CONFIGURATION_WARNING: 				st_Variable:= IotExtractType(monitor.battery.Events.b_CONFIGURATION_WARNING, 0, 0); 
// eDataMappingVarNames.battery_Events_b_POWERONFAULT: 				st_Variable:= IotExtractType(monitor.battery.Events.b_POWERONFAULT, 0, 0); 
// eDataMappingVarNames.battery_Events_b_POWEROFFFAULT: 				st_Variable:= IotExtractType(monitor.battery.Events.b_POWEROFFFAULT, 0, 0); 
// eDataMappingVarNames.battery_Events_b_DISCONNECTOR_OFF: 				st_Variable:= IotExtractType(monitor.battery.Events.b_DISCONNECTOR_OFF, 0, 0); 
// eDataMappingVarNames.battery_Events_b_SocLowLimitOutOfRange: 				st_Variable:= IotExtractType(monitor.battery.Events.b_SocLowLimitOutOfRange, 0, 0); 
// eDataMappingVarNames.battery_Events_b_SocHighLimitOutOfRange: 				st_Variable:= IotExtractType(monitor.battery.Events.b_SocHighLimitOutOfRange, 0, 0); 
// eDataMappingVarNames.battery_Events_b_SBMUCommError_0: 				st_Variable:= IotExtractType(monitor.battery.Events.b_SBMUCommError[0], 0, 0); 
// eDataMappingVarNames.battery_Events_b_SBMUCommError_1: 				st_Variable:= IotExtractType(monitor.battery.Events.b_SBMUCommError[1], 0, 0); 
// eDataMappingVarNames.battery_Events_b_SBMUCommError_2: 				st_Variable:= IotExtractType(monitor.battery.Events.b_SBMUCommError[2], 0, 0); 
// eDataMappingVarNames.battery_Events_b_SBMUCommError_3: 				st_Variable:= IotExtractType(monitor.battery.Events.b_SBMUCommError[3], 0, 0); 
// eDataMappingVarNames.battery_Events_b_SBMUFailedToConnect_0: 				st_Variable:= IotExtractType(monitor.battery.Events.b_SBMUFailedToConnect[0], 0, 0); 
// eDataMappingVarNames.battery_Events_b_SBMUFailedToConnect_1: 				st_Variable:= IotExtractType(monitor.battery.Events.b_SBMUFailedToConnect[1], 0, 0); 
// eDataMappingVarNames.battery_Events_b_SBMUFailedToConnect_2: 				st_Variable:= IotExtractType(monitor.battery.Events.b_SBMUFailedToConnect[2], 0, 0); 
// eDataMappingVarNames.battery_Events_b_SBMUFailedToConnect_3: 				st_Variable:= IotExtractType(monitor.battery.Events.b_SBMUFailedToConnect[3], 0, 0); 
// eDataMappingVarNames.protections_FireDetection_b_FireAlarm: 				st_Variable:= IotExtractType(monitor.protections.FireDetection.b_FireAlarm, 0, 0); 
// eDataMappingVarNames.protections_FireDetection_SmokeDetectors_State: 				st_Variable:= IotExtractType(monitor.protections.FireDetection.SmokeDetectors.State, 0, 0); 
// eDataMappingVarNames.protections_FireDetection_CODetectors_State: 				st_Variable:= IotExtractType(monitor.protections.FireDetection.CODetectors.State, 0, 0); 
// eDataMappingVarNames.protections_FireDetection_CODetectors_b_CoValuesOK: 				st_Variable:= IotExtractType(monitor.protections.FireDetection.CODetectors.b_CoValuesOK, 0, 0); 
// eDataMappingVarNames.protections_FireDetection_CODetectors_Value_0: 				st_Variable:= IotExtractType(monitor.protections.FireDetection.CODetectors.Value[0], 1, 0); 
// eDataMappingVarNames.protections_FireDetection_CODetectors_Value_1: 				st_Variable:= IotExtractType(monitor.protections.FireDetection.CODetectors.Value[1], 1, 0); 
// eDataMappingVarNames.protections_FireDetection_CODetectors_Value_2: 				st_Variable:= IotExtractType(monitor.protections.FireDetection.CODetectors.Value[2], 1, 0); 
// eDataMappingVarNames.protections_FireDetection_CODetectors_Value_3: 				st_Variable:= IotExtractType(monitor.protections.FireDetection.CODetectors.Value[3], 1, 0); 
// eDataMappingVarNames.protections_FireDetection_Events_CODetFault: 				st_Variable:= IotExtractType(monitor.protections.FireDetection.Events.CODetFault, 0, 0); 
// eDataMappingVarNames.protections_FireDetection_Events_CODetWarning1: 				st_Variable:= IotExtractType(monitor.protections.FireDetection.Events.CODetWarning1, 0, 0); 
// eDataMappingVarNames.protections_FireDetection_Events_CODetWarning2: 				st_Variable:= IotExtractType(monitor.protections.FireDetection.Events.CODetWarning2, 0, 0); 
// eDataMappingVarNames.protections_FireDetection_Events_CODetAlarm: 				st_Variable:= IotExtractType(monitor.protections.FireDetection.Events.CODetAlarm, 0, 0); 
// eDataMappingVarNames.protections_FireDetection_Events_SmokeDetFault: 				st_Variable:= IotExtractType(monitor.protections.FireDetection.Events.SmokeDetFault, 0, 0); 
// eDataMappingVarNames.protections_FireDetection_Events_SmokeDetAlarm: 				st_Variable:= IotExtractType(monitor.protections.FireDetection.Events.SmokeDetAlarm, 0, 0); 
// eDataMappingVarNames.protections_FireDetection_Events_AlarmMuted: 				st_Variable:= IotExtractType(monitor.protections.FireDetection.Events.AlarmMuted, 0, 0); 
// eDataMappingVarNames.protections_Insulation_b_Enabled: 				st_Variable:= IotExtractType(monitor.protections.Insulation.b_Enabled, 0, 0); 
// eDataMappingVarNames.protections_Insulation_b_PENlinkDetected: 				st_Variable:= IotExtractType(monitor.protections.Insulation.b_PENlinkDetected, 0, 0); 
// eDataMappingVarNames.protections_Insulation_b_Warning: 				st_Variable:= IotExtractType(monitor.protections.Insulation.b_Warning, 0, 0); 
// eDataMappingVarNames.protections_Insulation_e_EarthingSystemDetected: 				st_Variable:= IotExtractType(monitor.protections.Insulation.e_EarthingSystemDetected, 0, 0); 
// eDataMappingVarNames.protections_Insulation_b_PENlinkOperatedFault: 				st_Variable:= IotExtractType(monitor.protections.Insulation.b_PENlinkOperatedFault, 0, 0); 
// eDataMappingVarNames.protections_Insulation_b_EarthingSystemMismatch: 				st_Variable:= IotExtractType(monitor.protections.Insulation.b_EarthingSystemMismatch, 0, 0); 
// eDataMappingVarNames.protections_Insulation_b_NoEarthingSystemSet: 				st_Variable:= IotExtractType(monitor.protections.Insulation.b_NoEarthingSystemSet, 0, 0); 
// eDataMappingVarNames.protections_MRCDB_b_prewarning: 				st_Variable:= IotExtractType(monitor.protections.MRCDB.b_prewarning, 0, 0); 
// eDataMappingVarNames.protections_Surge_b_Type12_OK: 				st_Variable:= IotExtractType(monitor.protections.Surge.b_Type12_OK, 0, 0); 
// eDataMappingVarNames.protections_Surge_b_Type3_OK: 				st_Variable:= IotExtractType(monitor.protections.Surge.b_Type3_OK, 0, 0); 
// eDataMappingVarNames.protections_OvercurrentProtection_r_TotalOutputCurrentLimit: 				st_Variable:= IotExtractType(monitor.protections.OvercurrentProtection.r_TotalOutputCurrentLimit, 0, 0); 
// eDataMappingVarNames.protections_OvercurrentProtection_r_TotalInputCurrentLimit: 				st_Variable:= IotExtractType(monitor.protections.OvercurrentProtection.r_TotalInputCurrentLimit, 0, 0); 
// eDataMappingVarNames.protections_OvercurrentProtection_b_OutputWarning: 				st_Variable:= IotExtractType(monitor.protections.OvercurrentProtection.b_OutputWarning, 0, 0); 
// eDataMappingVarNames.protections_OvercurrentProtection_b_InputWarning: 				st_Variable:= IotExtractType(monitor.protections.OvercurrentProtection.b_InputWarning, 0, 0); 
// eDataMappingVarNames.protections_OvercurrentProtection_b_OutputAlarm: 				st_Variable:= IotExtractType(monitor.protections.OvercurrentProtection.b_OutputAlarm, 0, 0); 
// eDataMappingVarNames.protections_OvercurrentProtection_b_InputAlarm: 				st_Variable:= IotExtractType(monitor.protections.OvercurrentProtection.b_InputAlarm, 0, 0); 
// eDataMappingVarNames.protections_OvercurrentProtection_r_PeakCurrent: 				st_Variable:= IotExtractType(monitor.protections.OvercurrentProtection.r_PeakCurrent, 0, 0); 
// eDataMappingVarNames.protections_OvercurrentProtection_t_PeakCurrentDuration: 				st_Variable:= IotExtractType(monitor.protections.OvercurrentProtection.t_PeakCurrentDuration, 0, 0); 
// eDataMappingVarNames.protections_OvercurrentProtection_s_locationPeak: 				st_Variable:= IotExtractType(monitor.protections.OvercurrentProtection.s_locationPeak, 0, 0); 
// eDataMappingVarNames.peakshavebox_PSBmode: 				st_Variable:= IotExtractType(monitor.peakshavebox.PSBmode, 0, 0); 
// eDataMappingVarNames.peakshavebox_Powermonitor_ar_ApparentPower_AVG: 				st_Variable:= IotExtractType(monitor.peakshavebox.Powermonitor.ar_ApparentPower[0], 1, 1); 
